(* CoDeSys 2.3.9.55 project: tmeiccoolingskidv2.pro *)
(* Libraries: Standard.lib 20.5.14 01:13:26, Iecsfc.lib 30.1.13 06:05:12, SYSLIBCALLBACK.LIB 30.1.13 06:05:12 *)

(* PLC configuration (modules and I/O channels)
xWaterLow AT %IX10.0 [BOOLOnX_I] Ch_1 Digital input
xWaterLowLow AT %IX10.1 [BOOLOnX_I] Ch_2 Digital input
AT %IX10.2 [BOOLOnX_I] Ch_1 Digital input
AT %IX10.3 [BOOLOnX_I] Ch_2 Digital input
AT %IX10.4 [BOOLOnX_I] Ch_3 Digital input
AT %IX10.5 [BOOLOnX_I] Ch_4 Digital input
0750-0402 4 DI 24 V DC 3.0ms [Type_1_4_Channels] node 2, in %IX10.2 out %QB4
  AT %IX10.6 [BOOLOnX_I] Ch_1 Digital input
  AT %IX10.7 [BOOLOnX_I] Ch_2 Digital input
  AT %IX10.8 [BOOLOnX_I] Ch_3 Digital input
  AT %IX10.9 [BOOLOnX_I] Ch_4 Digital input
xOutput8DO1 AT %QX2.0 [BOOLOnX_Q] Ch_1 Digital output
AT %QX2.1 [BOOLOnX_Q] Ch_2 Digital output
AT %QX2.2 [BOOLOnX_Q] Ch_3 Digital output
AT %QX2.3 [BOOLOnX_Q] Ch_4 Digital output
AT %QX2.4 [BOOLOnX_Q] Ch_5 Digital output
AT %QX2.5 [BOOLOnX_Q] Ch_6 Digital output
AT %QX2.6 [BOOLOnX_Q] Ch_7 Digital output
AT %QX2.7 [BOOLOnX_Q] Ch_8 Digital output
xOutput AT %QX2.8 [BOOLOnX_Q] Ch_1 Digital output
AT %QX2.9 [BOOLOnX_Q] Ch_2 Digital output
AT %QX2.10 [BOOLOnX_Q] Ch_1 Digital output
AT %QX2.11 [BOOLOnX_Q] Ch_2 Digital output
0750-0492 2 AI 4-20mA Diff Measurement Input [Type_8_2_Channels] node 6, in %IB20 out %QB0
  AT %IW0 [WORDOnW_I] Ch_1 Input word
  AT %IW1 [WORDOnW_I] Ch_2 Input word
0750-0461 2 AI PT100 (RTD) [Type_44_2_Channels] node 7, in %IB20 out %QB0
  AT %IW2 [INTOnW_I] Ch_1 signed Input value
  AT %IW3 [INTOnW_I] Ch_2 signed Input value
0750-0461 2 AI PT100 (RTD) [Type_44_2_Channels] node 8, in %IB24 out %QB0
  AT %IW4 [INTOnW_I] Ch_1 signed Input value
  AT %IW5 [INTOnW_I] Ch_2 signed Input value
0750-0455 4 AI 4-20mA s.e. [Type_8_4_Channels] node 9, in %IB28 out %QB0
  AT %IW6 [WORDOnW_I] Ch_1 Input word
  AT %IW7 [WORDOnW_I] Ch_2 Input word
  AT %IW8 [WORDOnW_I] Ch_3 Input word
  AT %IW9 [WORDOnW_I] Ch_4 Input word
0750-0554 2 AO 4-20mA [Type_14_2_Channels] node 10, in %IB32 out %QB0
  AT %QW0 [WORDOnW_Q] Ch_1 Analog output
  AT %QW1 [WORDOnW_Q] Ch_2 Analog output
AT %IX10.10 [BOOLOnX_I] Ch_1 Digital input
AT %IX10.11 [BOOLOnX_I] Ch_2 Digital input
AT %IX10.12 [BOOLOnX_I] Ch_3 Digital input
AT %IX10.13 [BOOLOnX_I] Ch_4 Digital input
Modbus variables [PFC200MODBUS] node 1, in %IB0 out %QB0 {PlcStopBehaviour = 1; FiledbusErrorBehaviour = 1; TcpOperation = 1; TcpPort = 502; TcpTimeout = 600; UdpOperation = 1; UdpPort = 502; RtuOperation = 0; NodeId = 1; ResponseTimeout = 100; Interface = 0; Baud = 115200; StopBits = 1; Parity = 1; FlowCtrl = 0; PhysInterface = 0}
Modbus-Master [MB_MASTER] node 2, in %IB0 out %QB0
*)

(* Global variable list: Global_Variables *)
VAR_GLOBAL
	gaPumps: ARRAY [1..2] OF  ST_PUMP;
	gaTemps: ARRAY [1..3] OF ST_RTD;
	gaSwitches: ARRAY [1..3] OF ST_SWITCH;
	gaFans: ARRAY [1..4] OF ST_FAN;
	gConductivity: ST_COND;
	gFlow: ST_FLOW;
	gAct: ST_ACT;
	gSystem: ST_SYSTEM;
	gcAlarm: INT :=  1;
	gcFault:  INT := 0;
	gTempValCtrlSys: ST_TempValCtrlSys;
	gProgramErrors: ST_ProgramErrors;
	tbFailure: BOOL;
	tbSuccess: BOOL;
	tbTBLog: STRING(256);

	activePump: ST_PUMP;
	standbyPump: ST_PUMP;


END_VAR

(* Data type *)
TYPE HERE :
STRUCT
	On: BOOL;
	Off: BOOL;
	Fault: BOOL;
	Shutting_Down: BOOL;
	Initializing: BOOL;
	Calibrating: BOOL;
	Acknowledge_Fault: BOOL;
	LIST_FLAGS: ARRAY [1..25] OF BOOL;
	System_Active: BOOL;
	PA: BOOL;
	SA: BOOL;

END_STRUCT
END_TYPE

(* Data type in Instrument Data Types *)
TYPE RAWINPUT :
STRUCT
	wRawAnalogWord: WORD;
	iRawAnalogInt: INT;
	xRawDigital: BOOL;
END_STRUCT
END_TYPE

(* Data type *)
TYPE SignalIO :
STRUCT
END_STRUCT
END_TYPE

(* Data type *)
TYPE ST_ACT :
STRUCT
	stDescription: ST_Description;
	stActualization: ST_Analog;
	stCounters: ST_LGCount;
	stCalibrationStatus: ST_CalTest;
	rOpenPerc: REAL; (*Percentage of it being Open*)
END_STRUCT
END_TYPE

(* Data type *)
TYPE ST_ActivePumpStandbyPump :
STRUCT
END_STRUCT
END_TYPE

(* Data type *)
TYPE ST_Analog :
STRUCT
	rGain: REAL;
	rOffset: REAL;
	iRaw: REAL;
	rProcessed: REAL;
END_STRUCT
END_TYPE

(* Data type *)
TYPE ST_Backup :
STRUCT
	xActive: BOOL;
	xRedundant: BOOL;
END_STRUCT
END_TYPE

(* Data type *)
TYPE ST_CalTest :
STRUCT
	xCalibrated: BOOL;
	xTested: BOOL;
END_STRUCT
END_TYPE

(* Data type *)
TYPE ST_COND :
STRUCT
	stDescription: ST_Description;
	stConductivity: ST_Analog; (*Cond Reading Power*)
	stFault: ST_Digital; (*Fault Y/N*)
	stAlarm: ST_DIgital; (*Alarm Y/N*)
	stCounters: ST_LGCount;
	stCalibrationStatus: ST_CalTest;
END_STRUCT
END_TYPE

(* Data type *)
TYPE ST_Count :
STRUCT
	iAlarm: INT;
	iFault: INT;
	iForce: INT;
	iCalibrate: INT;
	iTest: INT;
END_STRUCT
END_TYPE

(* Data type *)
TYPE ST_Description :
STRUCT
	iID : INT;
	iState: INT; (*Offline, Standby,  Active, Calibration, Testing *)
	xFault: BOOL;
	xAlarm: BOOL;
	sDetail:  STRING;
END_STRUCT
END_TYPE

(* Data type *)
TYPE ST_Digital :
STRUCT
	iValue: INT;
END_STRUCT
END_TYPE

(* Data type *)
TYPE ST_FA :
STRUCT
	xFault: BOOL;
	xAlarm: BOOL;
END_STRUCT
END_TYPE

(* Data type *)
TYPE ST_FAN :
STRUCT
	stDescription: ST_Description;
	stActivate: ST_Digital; (*Pump On/Off*)
	stCounters: ST_LGCount;
	stCalibrationStatus: ST_CalTest;
	stBackup: ST_Backup;
END_STRUCT
END_TYPE

(* Data type *)
TYPE ST_FLOW :
STRUCT
	stDescription: ST_Description;
	stFlowRate: ST_Analog; (*Switch Trip*)
	stCounters: ST_LGCount;
	stCalibrationStatus: ST_CalTest;
END_STRUCT
END_TYPE

(* Data type *)
TYPE ST_HeartBeat :
STRUCT
	stDescription: ST_Description;
END_STRUCT
END_TYPE

(* Data type in Instrument Data Types *)
TYPE ST_INST :
STRUCT
	axBoolValues: ARRAY [1..10] OF BOOL;
	aiIntValues: ARRAY [1..10] OF REAL;

END_STRUCT
END_TYPE

(* Data type in Instrument Data Types *)
TYPE ST_INSTRUMENT :
STRUCT
	iState: INT; (*0 = Standby; 1 = Data Loading;*)
	stInput: ST_IO;
	stOutput: ST_IO;
	stMeasurement: ST_MEASUREMENTS;
	stActuateValues: ST_MEASUREMENTS;
END_STRUCT
END_TYPE

(* Data type in Flags *)
TYPE ST_InstrumentFlags :
STRUCT
	xConductivitySensorAlarmTrip: BOOL := FALSE;
	xConductivitySensorFaultTrip: BOOL := FALSE;
	xPump1BadRead: BOOL := FALSE;
	xPump2BadRead: BOOL := FALSE;
	xPump1LPError: BOOL := FALSE;
	xPump2LPError: BOOL := FALSE;
	xConductivitySensorBadRead: BOOL := FALSE;
	xConductivitySensorMisalignment: BOOL := FALSE;
	xConductivitySensorError: BOOL := FALSE;
	xFlowSensorBadRead: BOOL := FALSE;
	xRTD1BadRead: BOOL := FALSE;
	xRTD2BadRead: BOOL := FALSE;
	xRTD3BadRead: BOOL := FALSE;
	xNoPumpBackup: BOOL := FALSE;
	xPump1Failure: BOOL := FALSE;
	xPump2Failure: BOOL := FALSE;
	xRTD1Failure: BOOL := FALSE;
	xRTD2Failure: BOOL := FALSE;
	xRTD3Failure: BOOL := FALSE;
	xConductivitySensorFailure: BOOL := FALSE;
	xFlowSensorFailure: BOOL := FALSE;
	xPressureLow: BOOL := FALSE;
	xPumpPowerLow: BOOL := FALSE;
	xFlowLow: BOOL := FALSE;
	xWaterLevelSensorError: BOOL := FALSE;
END_STRUCT
END_TYPE

(* Data type *)
TYPE ST_IO :
STRUCT
	axDigital: ARRAY [1..100] OF BOOL;
	awAnalog: ARRAY[1..100] OF WORD;
	aiAnalog: ARRAY[1..100] OF INT;
END_STRUCT
END_TYPE

(* Data type *)
TYPE ST_LGCount :
STRUCT
	stLocal : ST_Count;
	stGlobal: ST_Count;
END_STRUCT
END_TYPE

(* Data type in Instrument Data Types *)
TYPE ST_MEASUREMENTS :
STRUCT
	axDigital: ARRAY [1..100] OF BOOL;
	arAnalog: ARRAY[1..100] OF REAL;
END_STRUCT
END_TYPE

(* Data type *)
TYPE ST_PRES :
STRUCT
	stDescription: ST_Description;
	stSwitchTrip: ST_Digital; (*Switch Trip*)
	stCounters: ST_LGCount;
	stCalibrationStatus: ST_CalTest;
END_STRUCT
END_TYPE

(* Data type *)
TYPE ST_ProgramErrors :
STRUCT
	xTempValCtrlSys: BOOL;
	xDataConversion: BOOL;
END_STRUCT
END_TYPE

(* Data type *)
TYPE ST_PUMP :
STRUCT
	stDescription: ST_Description;
	stPumpPower: ST_Analog; (*Pump Power*)
	stActivate: ST_Digital; (*Pump On/Off*)
	stCounters: ST_LGCount;
	stCalibrationStatus: ST_CalTest;
	stBackup: ST_Backup;
END_STRUCT
END_TYPE

(* Data type *)
TYPE ST_RTD :
STRUCT
	stDescription: ST_Description;
	stTempRead: ST_Analog;
	stCounters: ST_LGCount;
	stCalibrationStatus: ST_CalTest;
END_STRUCT
END_TYPE

(* Data type *)
TYPE ST_SPT :
STRUCT
	rSetpoint: REAL;
	rThreshold: REAL;
END_STRUCT
END_TYPE

(* Data type *)
TYPE ST_SWITCH :
STRUCT
	stDescription: ST_Description;
	stSwitchTrip: ST_Digital; (*Switch Trip*)
	stCounters: ST_LGCount;
	stCalibrationStatus: ST_CalTest;
END_STRUCT
END_TYPE

(* Data type *)
TYPE ST_SYSTEM :
STRUCT
	stSystemCounters: ST_SystemCounters;
	stSystemFlags: ST_SystemFlags;
	stInstrumentFlags: ST_instrumentFlags;
	stInputs: ST_SystemInputs;
	stOutputs: ST_SystemOutputs;
END_STRUCT
END_TYPE

(* Data type *)
TYPE ST_SystemCounters :
STRUCT
	iRTDFailures: INT;
	iPumpFailures: INT;
	iActivePump: INT;
	iActiveFanGroup: INT;
END_STRUCT
END_TYPE

(* Data type *)
TYPE ST_SystemFlags :
STRUCT
	xSwitchPumpRequest: BOOL;
	xAwaitInitialization: BOOL;
	xAwaitCalibration: BOOL;
	xFault: BOOL;
	xAlarm: BOOL;
	xPPFError: BOOL;
	xWaterLow: BOOL;
	xWaterVeryLow: BOOL;
END_STRUCT
END_TYPE

(* Data type *)
TYPE ST_SystemInputs :
STRUCT
	rPumpPower: REAL;
	rFlowRate: REAL;
	rConductivity: REAL;
	rTemperature: REAL;
	xPressureLow: BOOL;
	xWaterLow: BOOL;
	xWaterLowLow: BOOL;
	xSystemON: BOOL;
	xConductivityAlarm: BOOL;
	xConductivityFault: BOOL;
END_STRUCT
END_TYPE

(* Data type *)
TYPE ST_SystemMeasurement :
STRUCT

END_STRUCT
END_TYPE

(* Data type *)
TYPE ST_SystemOutputs :
STRUCT
	rValveActuate: REAL;
	xPump1Activate: BOOL;
	xPump2Activate: BOOL;
	xFan12Activate: BOOL;
	xFan34Activate: BOOL;
END_STRUCT
END_TYPE

(* Data type *)
TYPE ST_TempValCtrlSys :
STRUCT
	rDiffThresh: REAL;
	rDiffTol: REAL;
	iSysMeasState: INT;
	xFault: BOOL; (*Fault when all controlers are bad, or program error*)
	xAlarm: BOOL; (*Alarm for fault, when controller is bad, or program error*)
END_STRUCT
END_TYPE

(* POU PLC_PRG, LD *)
PROGRAM PLC_PRG
VAR PERSISTENT
	stPump1: ST_INSTRUMENT;
	stPump2: ST_INSTRUMENT;
	stPump3: ST_INSTRUMENT;
	stRTD1: ST_INSTRUMENT;
	stRTD2: ST_INSTRUMENT;
	stRTD3: ST_INSTRUMENT;
	stFan1: ST_INSTRUMENT;
	stFan2: ST_INSTRUMENT;
	stFan3: ST_INSTRUMENT;
	stFan4: ST_INSTRUMENT;
	stConductivitySensor: ST_INSTRUMENT;
	stFlowSensor: ST_INSTRUMENT;
	stWaterLevelLow: ST_INSTRUMENT;
	stWaterLevelLowLow: ST_INSTRUMENT;
	stPressureLowSensor: ST_INSTRUMENT;
	stSystemRunSwitch: ST_INSTRUMENT;

	stInstrumentFlags: ST_InstrumentFlags;

	stSystem: ST_SYSTEM;
END_VAR
VAR
		xReadAnalog: BOOL;
	xReadTemperature: BOOL;
	fbRunTestBench: RunTestBench;
	xTesting: BOOL;
	xReadDigital: BOOL;
	fbWaterLevelLowCaputer: FB_DigitalCapture;
	fbWaterLevelLowLowCapture: FB_DigitalCapture;
	fbConductivityAlarmCapture: FB_DigitalCapture;
	fbAssignAnalogValues: FB_AssignAnalog;
	fbAAP1: FB_AssignAnalog;
	fbAAP2: FB_AssignAnalog;
	fbAARTD1: FB_AssignAnalog;
	fbAARTD2: FB_AssignAnalog;
	fbAARTD3: FB_AssignAnalog;
	fbAAF3: FB_AssignAnalog;
	fbAAF: FB_AssignAnalog;
	fbAAC: FB_AssignAnalog;
END_VAR
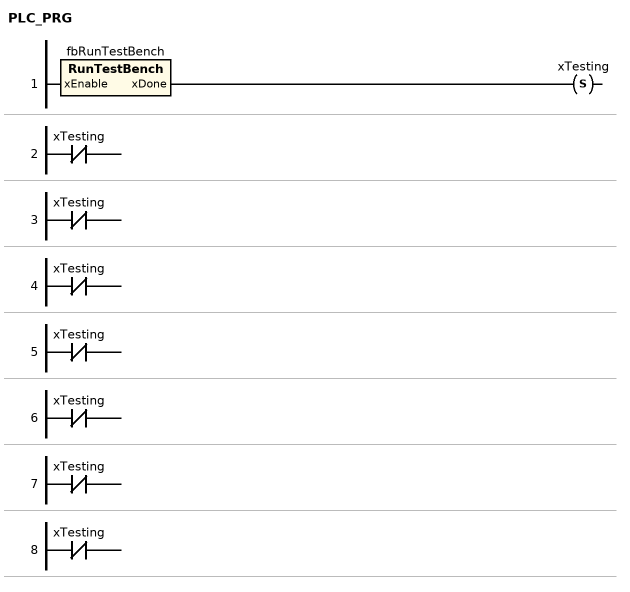
_LD_ (* Ladder Diagram *)
NETWORK 1
	fbRunTestBench:RunTestBench(xEnable: *) --- (S xTesting)
NETWORK 2
	[/xTesting]
NETWORK 3
	[/xTesting]
NETWORK 4
	[/xTesting]
NETWORK 5
	[/xTesting]
NETWORK 6
	[/xTesting]
NETWORK 7
	[/xTesting]
NETWORK 8
	[/xTesting]
_END_LD_
(* the same logic as Structured Text *)
(* Network 1 *)
fbRunTestBench(xEnable := TRUE);
IF fbRunTestBench.xDone THEN xTesting := TRUE; END_IF;
(* Network 2 *)
(* Network 3 *)
(* Network 4 *)
(* Network 5 *)
(* Network 6 *)
(* Network 7 *)
(* Network 8 *)
END_PROGRAM

(* POU RunTestBench, ST *)
FUNCTION_BLOCK RunTestBench
VAR_INPUT
	xEnable: BOOL;
END_VAR
VAR_OUTPUT
	xDone: BOOL := TRUE;
END_VAR
VAR
	istopCase: INT;
	iWait: INT := 0;
END_VAR
IF xEnable = FALSE THEN
	RETURN;
END_IF
TB_MainProgram2();
END_FUNCTION_BLOCK

(* POU TB_MainProgram2, LD *)
PROGRAM TB_MainProgram2
VAR
	PUMP1: ST_INSTRUMENT;
	PUMP2: ST_INSTRUMENT;
	RTD1: ST_INSTRUMENT;
	RTD2: ST_INSTRUMENT;
	RTD3: ST_INSTRUMENT;
	CONDUCTIVITY: ST_INSTRUMENT;
	FLOW: ST_INSTRUMENT;
	WATERLOW: ST_INSTRUMENT;
	WATERLOWLOW: ST_INSTRUMENT;
	PRESSURELOW: ST_INSTRUMENT;
	SYSTEM: ST_SYSTEM;
	main: HERE;
	p1i: WORD := 32768;
	p2i: WORD := 50;
	t1i: INT := 100;
	t2i: INT:= 100;
	t3i: INT:= 100;
	fi: WORD:= 50;
	ci: WORD:= 40;
	wli: BOOL:= FALSE;
	wlli: BOOL:= FALSE;
	cai: BOOL:= FALSE;
	cfi: BOOL:= FALSE;
	pli: BOOL:= FALSE;
	p1mas: REAL:= 32767;
	p2mas: REAL:= 32767;
	t1mas: REAL:= 32767;
	t2mas: REAL:= 32767;
	t3mas: REAL:= 32767;
	fmas: REAL:= 32767;
	cmas: REAL:= 32767;
	p1mis: REAL:= -32768;
	p2mis: REAL:= -32768;
	t1mis: REAL:= 0;
	t2mis: REAL:= 0;
	t3mis: REAL:= 0;
	fmis: REAL:= -32768;
	cmis: REAL:= -32768;
	p1mav: REAL:= 55;
	p2mav: REAL:= 55;
	t1mav: REAL:= 100;
	t2mav: REAL:= 100;
	t3mav: REAL:= 100;
	fmav: REAL:= 20;
	cmaV: REAL:= 2000;
	p1miv: REAL:= 0;
	p2miv: REAL:= 0;
	t1miv: REAL:= 0;
	t2miv: REAL:= 0;
	t3miv: REAL:= 0;
	fmiv: REAL:= 0;
	cmiv: REAL:= 2;
	p1tol: REAL:= 0;
	p2tol: REAL:= 0;
	t1tol: REAL:= 0;
	t2tol: REAL:= 0;
	t3tol: REAL:= 0;
	ftol: REAL:= 0;
	ctol: REAL:=0;
	p1t: TIME:= T#100MS;
	p2t: TIME:= T#100MS;
	t1t: TIME:= T#100MS;
	t2t: TIME:= T#100MS;
	t3t: TIME:= T#100MS;
	ft: TIME:= T#100MS;
	ct: TIME:= T#100MS;
	wlt: TIME:= T#100MS;
	wllt: TIME:= T#100MS;
	cat: TIME:= T#100MS;
	cft: TIME:= T#100MS;
	plt: TIME:= T#100MS;

	p1o: BOOL;
	p2o: BOOL;
	t1o: BOOL;
	t2o: BOOL;
	t3o: BOOL;
	fo: BOOL;
	co: BOOL;
	wlo: BOOL;
	wllo: BOOL;
	cao: BOOL;
	cfo: BOOL;
	plo: BOOL;
	dummy: BOOL;
	fbinstrumentinputscan: FB_InstrumentInputScan;
	fbsysteminstrumentalignment: FB_SystemInstrumentAlignment;
	fbcheckwaterlevel: FB_CheckWaterLevel;
	fbcheckconductivity: FB_CheckConductivity;
	fbpowerpressureflowthreshold: FB_PowerPressureFlowThreshold;
	fbpowerpressureflowvote: FB_PowerPressureFlowVote;
	fbpumpstartswitchroutine: FB_PumpStartSwitchRoutine;
	xsysalrm1: BOOL;
	xsysfault1: BOOL;
	xsysalarm2: BOOL;
	xsysfault3: BOOL;
	xsysfault2: BOOL;
		xsysalarm3: BOOL;
		xsysalarm4: BOOL;
		xsysfault4: BOOL;
		xpumpswitchrequest2: BOOL;
		xpumpswitchrequest1: BOOL;
		xSystemRun: BOOL;
		xStartDelay: BOOL;
		startdelaytimer: TON;
		fbtempboundcheck: FB_TemperatureBoundCheck;
		xsysalarm5: BOOL;
	xsysfault5: BOOL;
	fbsysstart: FB_SystemStart;
	fbfaultcheck: FB_FaultCheck;
	fbstop: FB_SystemStop;
	fbpumpcontrol: FB_PumpControl;
END_VAR
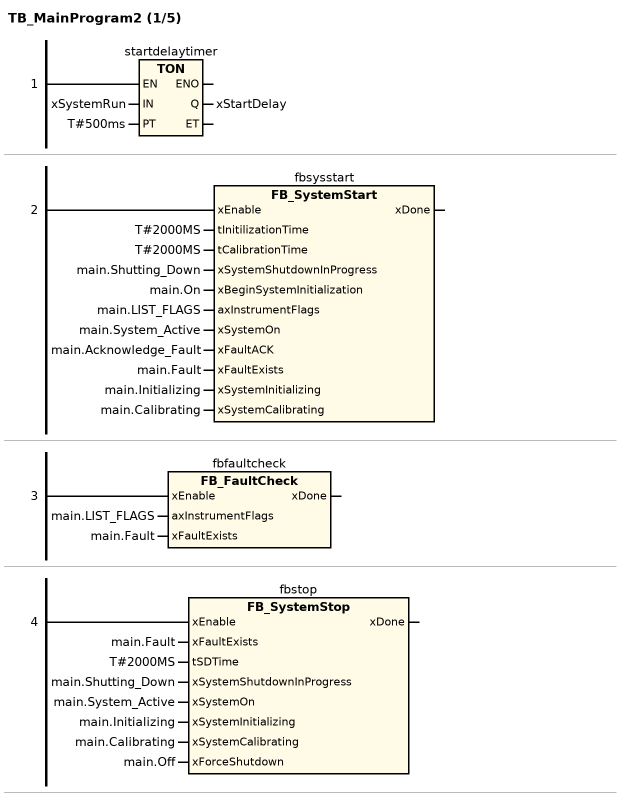
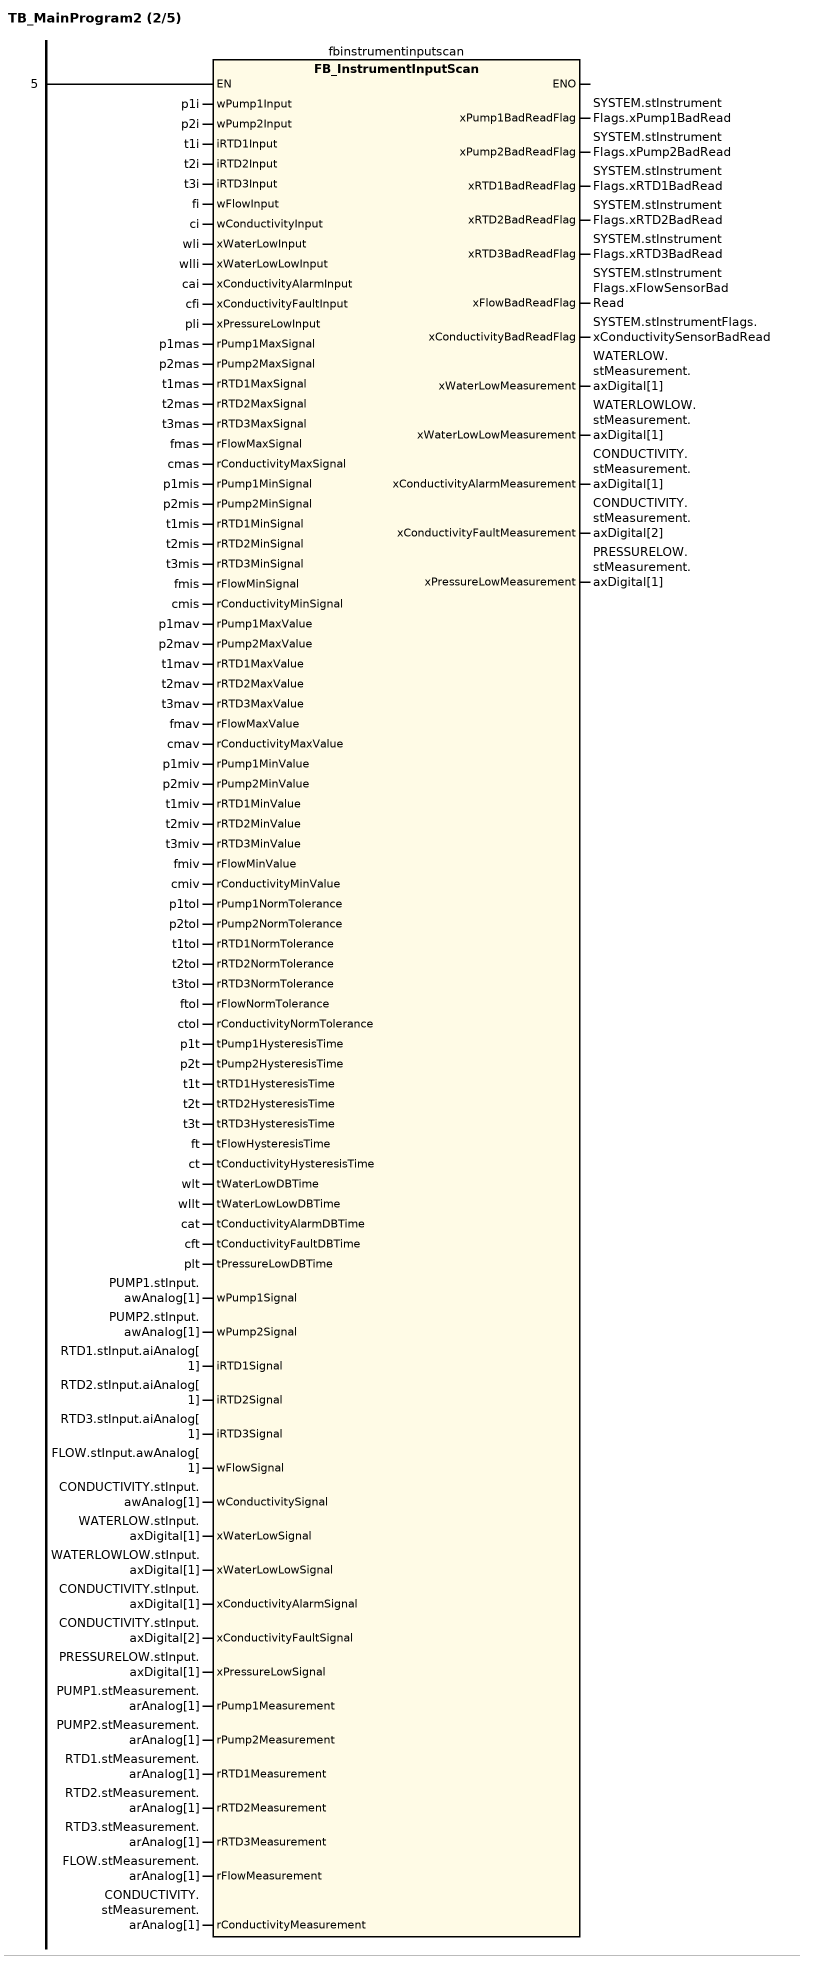
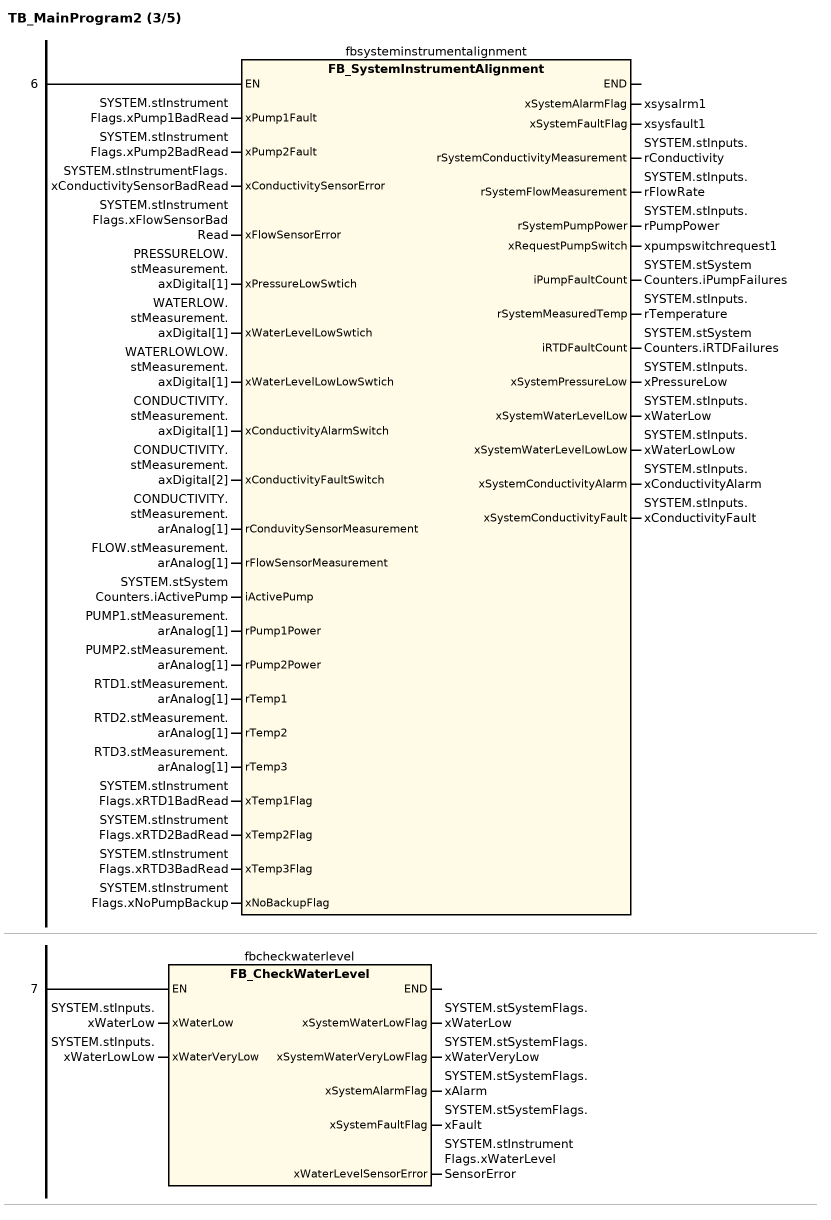
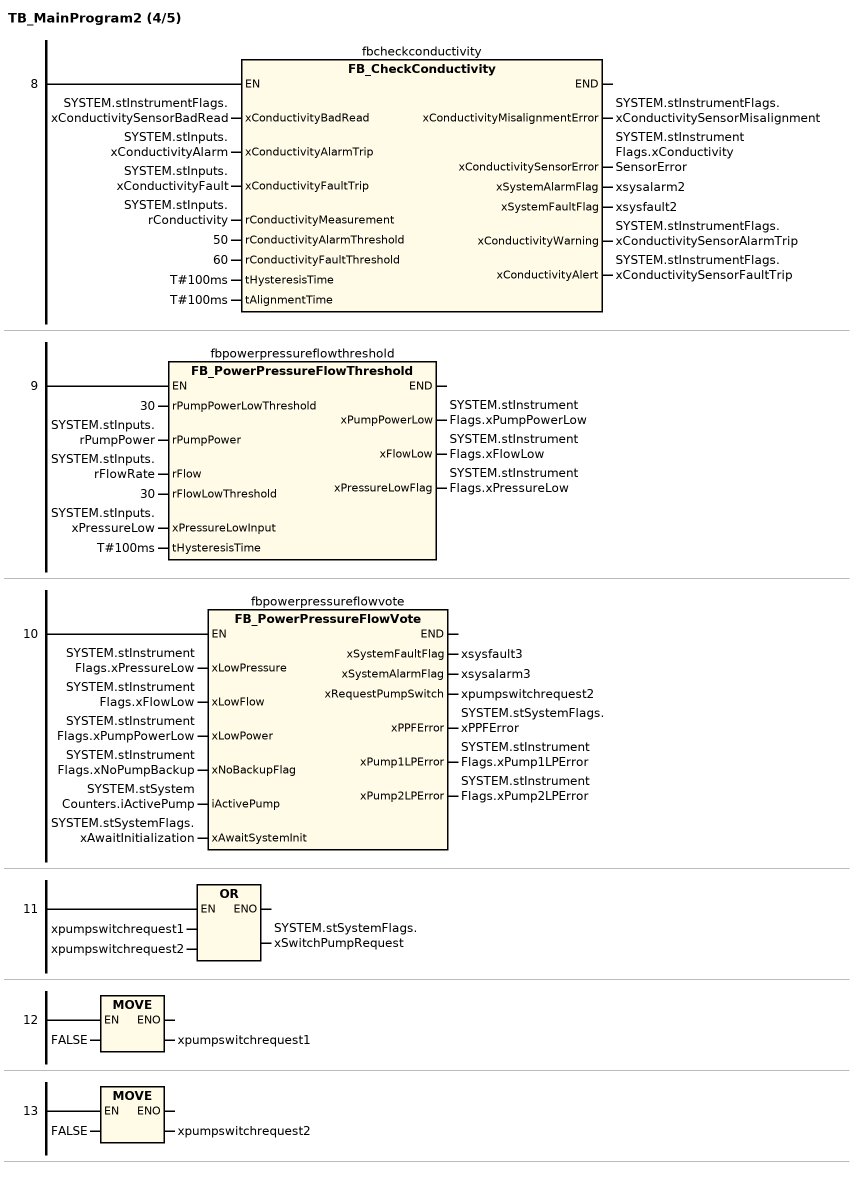
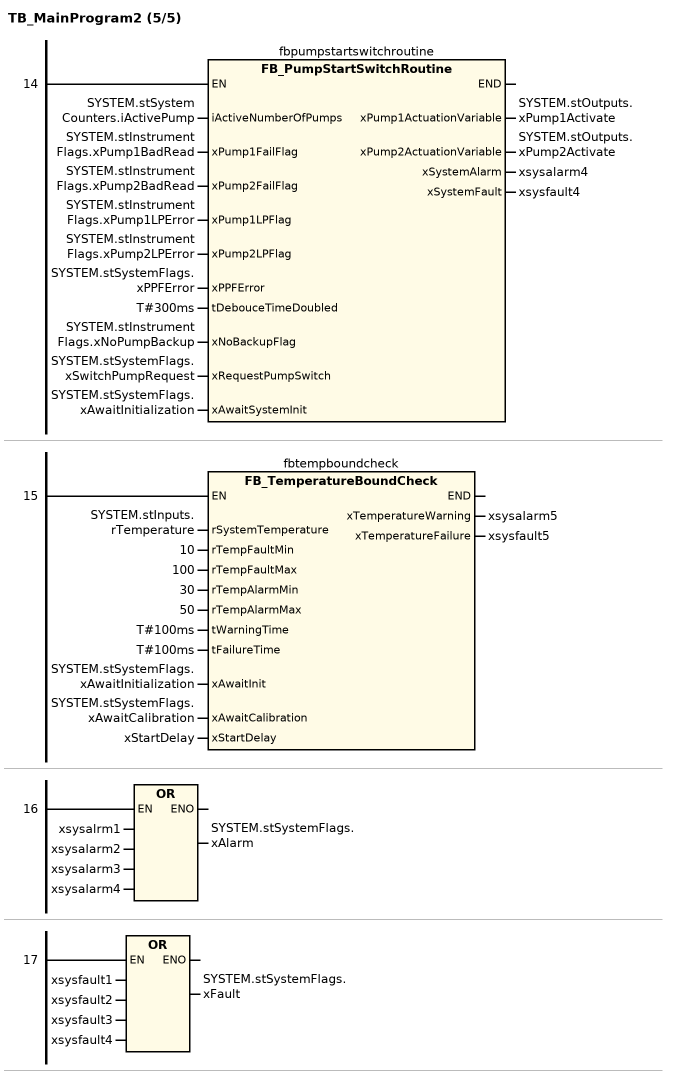
_LD_ (* Ladder Diagram *)
NETWORK 1
	*
		EN --- startdelaytimer:TON(IN: xSystemRun, PT: T#500ms) => xStartDelay
NETWORK 2
	fbsysstart:FB_SystemStart(xEnable: *, tInitilizationTime: T#2000MS, tCalibrationTime: T#2000MS, xSystemShutdownInProgress: main.Shutting_Down, xBeginSystemInitialization: main.On, axInstrumentFlags: main.LIST_FLAGS, xSystemOn: main.System_Active, xFaultACK: main.Acknowledge_Fault, xFaultExists: main.Fault, xSystemInitializing: main.Initializing, xSystemCalibrating: main.Calibrating)
NETWORK 3
	fbfaultcheck:FB_FaultCheck(xEnable: *, axInstrumentFlags: main.LIST_FLAGS, xFaultExists: main.Fault)
NETWORK 4
	fbstop:FB_SystemStop(xEnable: *, xFaultExists: main.Fault, tSDTime: T#2000MS, xSystemShutdownInProgress: main.Shutting_Down, xSystemOn: main.System_Active, xSystemInitializing: main.Initializing, xSystemCalibrating: main.Calibrating, xForceShutdown: main.Off)
NETWORK 5
	*
		EN --- fbinstrumentinputscan:FB_InstrumentInputScan(wPump1Input: p1i, wPump2Input: p2i, iRTD1Input: t1i, iRTD2Input: t2i, iRTD3Input: t3i, wFlowInput: fi, wConductivityInput: ci, xWaterLowInput: wli, xWaterLowLowInput: wlli, xConductivityAlarmInput: cai, xConductivityFaultInput: cfi, xPressureLowInput: pli, rPump1MaxSignal: p1mas, rPump2MaxSignal: p2mas, rRTD1MaxSignal: t1mas, rRTD2MaxSignal: t2mas, rRTD3MaxSignal: t3mas, rFlowMaxSignal: fmas, rConductivityMaxSignal: cmas, rPump1MinSignal: p1mis, rPump2MinSignal: p2mis, rRTD1MinSignal: t1mis, rRTD2MinSignal: t2mis, rRTD3MinSignal: t3mis, rFlowMinSignal: fmis, rConductivityMinSignal: cmis, rPump1MaxValue: p1mav, rPump2MaxValue: p2mav, rRTD1MaxValue: t1mav, rRTD2MaxValue: t2mav, rRTD3MaxValue: t3mav, rFlowMaxValue: fmav, rConductivityMaxValue: cmav, rPump1MinValue: p1miv, rPump2MinValue: p2miv, rRTD1MinValue: t1miv, rRTD2MinValue: t2miv, rRTD3MinValue: t3miv, rFlowMinValue: fmiv, rConductivityMinValue: cmiv, rPump1NormTolerance: p1tol, rPump2NormTolerance: p2tol, rRTD1NormTolerance: t1tol, rRTD2NormTolerance: t2tol, rRTD3NormTolerance: t3tol, rFlowNormTolerance: ftol, rConductivityNormTolerance: ctol, tPump1HysteresisTime: p1t, tPump2HysteresisTime: p2t, tRTD1HysteresisTime: t1t, tRTD2HysteresisTime: t2t, tRTD3HysteresisTime: t3t, tFlowHysteresisTime: ft, tConductivityHysteresisTime: ct, tWaterLowDBTime: wlt, tWaterLowLowDBTime: wllt, tConductivityAlarmDBTime: cat, tConductivityFaultDBTime: cft, tPressureLowDBTime: plt, wPump1Signal: PUMP1.stInput.awAnalog[1], wPump2Signal: PUMP2.stInput.awAnalog[1], iRTD1Signal: RTD1.stInput.aiAnalog[1], iRTD2Signal: RTD2.stInput.aiAnalog[1], iRTD3Signal: RTD3.stInput.aiAnalog[1], wFlowSignal: FLOW.stInput.awAnalog[1], wConductivitySignal: CONDUCTIVITY.stInput.awAnalog[1], xWaterLowSignal: WATERLOW.stInput.axDigital[1], xWaterLowLowSignal: WATERLOWLOW.stInput.axDigital[1], xConductivityAlarmSignal: CONDUCTIVITY.stInput.axDigital[1], xConductivityFaultSignal: CONDUCTIVITY.stInput.axDigital[2], xPressureLowSignal: PRESSURELOW.stInput.axDigital[1], rPump1Measurement: PUMP1.stMeasurement.arAnalog[1], rPump2Measurement: PUMP2.stMeasurement.arAnalog[1], rRTD1Measurement: RTD1.stMeasurement.arAnalog[1], rRTD2Measurement: RTD2.stMeasurement.arAnalog[1], rRTD3Measurement: RTD3.stMeasurement.arAnalog[1], rFlowMeasurement: FLOW.stMeasurement.arAnalog[1], rConductivityMeasurement: CONDUCTIVITY.stMeasurement.arAnalog[1], xPump2BadReadFlag => SYSTEM.stInstrumentFlags.xPump2BadRead, xRTD1BadReadFlag => SYSTEM.stInstrumentFlags.xRTD1BadRead, xRTD2BadReadFlag => SYSTEM.stInstrumentFlags.xRTD2BadRead, xRTD3BadReadFlag => SYSTEM.stInstrumentFlags.xRTD3BadRead, xFlowBadReadFlag => SYSTEM.stInstrumentFlags.xFlowSensorBadRead, xConductivityBadReadFlag => SYSTEM.stInstrumentFlags.xConductivitySensorBadRead, xWaterLowMeasurement => WATERLOW.stMeasurement.axDigital[1], xWaterLowLowMeasurement => WATERLOWLOW.stMeasurement.axDigital[1], xConductivityAlarmMeasurement => CONDUCTIVITY.stMeasurement.axDigital[1], xConductivityFaultMeasurement => CONDUCTIVITY.stMeasurement.axDigital[2], xPressureLowMeasurement => PRESSURELOW.stMeasurement.axDigital[1]) => SYSTEM.stInstrumentFlags.xPump1BadRead
NETWORK 6
	fbsysteminstrumentalignment:FB_SystemInstrumentAlignment(EN: *, xPump1Fault: SYSTEM.stInstrumentFlags.xPump1BadRead, xPump2Fault: SYSTEM.stInstrumentFlags.xPump2BadRead, xConductivitySensorError: SYSTEM.stInstrumentFlags.xConductivitySensorBadRead, xFlowSensorError: SYSTEM.stInstrumentFlags.xFlowSensorBadRead, xPressureLowSwtich: PRESSURELOW.stMeasurement.axDigital[1], xWaterLevelLowSwtich: WATERLOW.stMeasurement.axDigital[1], xWaterLevelLowLowSwtich: WATERLOWLOW.stMeasurement.axDigital[1], xConductivityAlarmSwitch: CONDUCTIVITY.stMeasurement.axDigital[1], xConductivityFaultSwitch: CONDUCTIVITY.stMeasurement.axDigital[2], rConduvitySensorMeasurement: CONDUCTIVITY.stMeasurement.arAnalog[1], rFlowSensorMeasurement: FLOW.stMeasurement.arAnalog[1], iActivePump: SYSTEM.stSystemCounters.iActivePump, rPump1Power: PUMP1.stMeasurement.arAnalog[1], rPump2Power: PUMP2.stMeasurement.arAnalog[1], rTemp1: RTD1.stMeasurement.arAnalog[1], rTemp2: RTD2.stMeasurement.arAnalog[1], rTemp3: RTD3.stMeasurement.arAnalog[1], xTemp1Flag: SYSTEM.stInstrumentFlags.xRTD1BadRead, xTemp2Flag: SYSTEM.stInstrumentFlags.xRTD2BadRead, xTemp3Flag: SYSTEM.stInstrumentFlags.xRTD3BadRead, xNoBackupFlag: SYSTEM.stInstrumentFlags.xNoPumpBackup, xSystemAlarmFlag => xsysalrm1, xSystemFaultFlag => xsysfault1, rSystemConductivityMeasurement => SYSTEM.stInputs.rConductivity, rSystemFlowMeasurement => SYSTEM.stInputs.rFlowRate, rSystemPumpPower => SYSTEM.stInputs.rPumpPower, xRequestPumpSwitch => xpumpswitchrequest1, iPumpFaultCount => SYSTEM.stSystemCounters.iPumpFailures, rSystemMeasuredTemp => SYSTEM.stInputs.rTemperature, iRTDFaultCount => SYSTEM.stSystemCounters.iRTDFailures, xSystemPressureLow => SYSTEM.stInputs.xPressureLow, xSystemWaterLevelLow => SYSTEM.stInputs.xWaterLow, xSystemWaterLevelLowLow => SYSTEM.stInputs.xWaterLowLow, xSystemConductivityAlarm => SYSTEM.stInputs.xConductivityAlarm, xSystemConductivityFault => SYSTEM.stInputs.xConductivityFault)
NETWORK 7
	fbcheckwaterlevel:FB_CheckWaterLevel(EN: *, xWaterLow: SYSTEM.stInputs.xWaterLow, xWaterVeryLow: SYSTEM.stInputs.xWaterLowLow, xSystemWaterLowFlag => SYSTEM.stSystemFlags.xWaterLow, xSystemWaterVeryLowFlag => SYSTEM.stSystemFlags.xWaterVeryLow, xSystemAlarmFlag => SYSTEM.stSystemFlags.xAlarm, xSystemFaultFlag => SYSTEM.stSystemFlags.xFault, xWaterLevelSensorError => SYSTEM.stInstrumentFlags.xWaterLevelSensorError)
NETWORK 8
	fbcheckconductivity:FB_CheckConductivity(EN: *, xConductivityBadRead: SYSTEM.stInstrumentFlags.xConductivitySensorBadRead, xConductivityAlarmTrip: SYSTEM.stInputs.xConductivityAlarm, xConductivityFaultTrip: SYSTEM.stInputs.xConductivityFault, rConductivityMeasurement: SYSTEM.stInputs.rConductivity, rConductivityAlarmThreshold: 50, rConductivityFaultThreshold: 60, tHysteresisTime: T#100ms, tAlignmentTime: T#100ms, xConductivityMisalignmentError => SYSTEM.stInstrumentFlags.xConductivitySensorMisalignment, xConductivitySensorError => SYSTEM.stInstrumentFlags.xConductivitySensorError, xSystemAlarmFlag => xsysalarm2, xSystemFaultFlag => xsysfault2, xConductivityWarning => SYSTEM.stInstrumentFlags.xConductivitySensorAlarmTrip, xConductivityAlert => SYSTEM.stInstrumentFlags.xConductivitySensorFaultTrip)
NETWORK 9
	fbpowerpressureflowthreshold:FB_PowerPressureFlowThreshold(EN: *, rPumpPowerLowThreshold: 30, rPumpPower: SYSTEM.stInputs.rPumpPower, rFlow: SYSTEM.stInputs.rFlowRate, rFlowLowThreshold: 30, xPressureLowInput: SYSTEM.stInputs.xPressureLow, tHysteresisTime: T#100ms, xPumpPowerLow => SYSTEM.stInstrumentFlags.xPumpPowerLow, xFlowLow => SYSTEM.stInstrumentFlags.xFlowLow, xPressureLowFlag => SYSTEM.stInstrumentFlags.xPressureLow)
NETWORK 10
	fbpowerpressureflowvote:FB_PowerPressureFlowVote(EN: *, xLowPressure: SYSTEM.stInstrumentFlags.xPressureLow, xLowFlow: SYSTEM.stInstrumentFlags.xFlowLow, xLowPower: SYSTEM.stInstrumentFlags.xPumpPowerLow, xNoBackupFlag: SYSTEM.stInstrumentFlags.xNoPumpBackup, iActivePump: SYSTEM.stSystemCounters.iActivePump, xAwaitSystemInit: SYSTEM.stSystemFlags.xAwaitInitialization, xSystemFaultFlag => xsysfault3, xSystemAlarmFlag => xsysalarm3, xRequestPumpSwitch => xpumpswitchrequest2, xPPFError => SYSTEM.stSystemFlags.xPPFError, xPump1LPError => SYSTEM.stInstrumentFlags.xPump1LPError, xPump2LPError => SYSTEM.stInstrumentFlags.xPump2LPError)
NETWORK 11
	*
		EN --- OR(xpumpswitchrequest1, xpumpswitchrequest2) => SYSTEM.stSystemFlags.xSwitchPumpRequest
NETWORK 12
	*
		EN --- MOVE(FALSE) => xpumpswitchrequest1
NETWORK 13
	*
		EN --- MOVE(FALSE) => xpumpswitchrequest2
NETWORK 14
	fbpumpstartswitchroutine:FB_PumpStartSwitchRoutine(EN: *, iActiveNumberOfPumps: SYSTEM.stSystemCounters.iActivePump, xPump1FailFlag: SYSTEM.stInstrumentFlags.xPump1BadRead, xPump2FailFlag: SYSTEM.stInstrumentFlags.xPump2BadRead, xPump1LPFlag: SYSTEM.stInstrumentFlags.xPump1LPError, xPump2LPFlag: SYSTEM.stInstrumentFlags.xPump2LPError, xPPFError: SYSTEM.stSystemFlags.xPPFError, tDebouceTimeDoubled: T#300ms, xNoBackupFlag: SYSTEM.stInstrumentFlags.xNoPumpBackup, xRequestPumpSwitch: SYSTEM.stSystemFlags.xSwitchPumpRequest, xAwaitSystemInit: SYSTEM.stSystemFlags.xAwaitInitialization, xPump1ActuationVariable => SYSTEM.stOutputs.xPump1Activate, xPump2ActuationVariable => SYSTEM.stOutputs.xPump2Activate, xSystemAlarm => xsysalarm4, xSystemFault => xsysfault4)
NETWORK 15
	fbtempboundcheck:FB_TemperatureBoundCheck(EN: *, rSystemTemperature: SYSTEM.stInputs.rTemperature, rTempFaultMin: 10, rTempFaultMax: 100, rTempAlarmMin: 30, rTempAlarmMax: 50, tWarningTime: T#100ms, tFailureTime: T#100ms, xAwaitInit: SYSTEM.stSystemFlags.xAwaitInitialization, xAwaitCalibration: SYSTEM.stSystemFlags.xAwaitCalibration, xStartDelay: xStartDelay, xTemperatureWarning => xsysalarm5, xTemperatureFailure => xsysfault5)
NETWORK 16
	*
		EN --- OR(xsysalrm1, xsysalarm2, xsysalarm3, xsysalarm4) => SYSTEM.stSystemFlags.xAlarm
NETWORK 17
	*
		EN --- OR(xsysfault1, xsysfault2, xsysfault3, xsysfault4) => SYSTEM.stSystemFlags.xFault
_END_LD_
(* the same logic as Structured Text *)
(* Network 1 *)
startdelaytimer(IN := xSystemRun, PT := T#500ms);
xStartDelay := startdelaytimer.Q;
(* Network 2 *)
fbsysstart(xEnable := TRUE, tInitilizationTime := T#2000MS, tCalibrationTime := T#2000MS, xSystemShutdownInProgress := main.Shutting_Down, xBeginSystemInitialization := main.On, axInstrumentFlags := main.LIST_FLAGS, xSystemOn := main.System_Active, xFaultACK := main.Acknowledge_Fault, xFaultExists := main.Fault, xSystemInitializing := main.Initializing, xSystemCalibrating := main.Calibrating);
(* Network 3 *)
fbfaultcheck(xEnable := TRUE, axInstrumentFlags := main.LIST_FLAGS, xFaultExists := main.Fault);
(* Network 4 *)
fbstop(xEnable := TRUE, xFaultExists := main.Fault, tSDTime := T#2000MS, xSystemShutdownInProgress := main.Shutting_Down, xSystemOn := main.System_Active, xSystemInitializing := main.Initializing, xSystemCalibrating := main.Calibrating, xForceShutdown := main.Off);
(* Network 5 *)
fbinstrumentinputscan(wPump1Input := p1i, wPump2Input := p2i, iRTD1Input := t1i, iRTD2Input := t2i, iRTD3Input := t3i, wFlowInput := fi, wConductivityInput := ci, xWaterLowInput := wli, xWaterLowLowInput := wlli, xConductivityAlarmInput := cai, xConductivityFaultInput := cfi, xPressureLowInput := pli, rPump1MaxSignal := p1mas, rPump2MaxSignal := p2mas, rRTD1MaxSignal := t1mas, rRTD2MaxSignal := t2mas, rRTD3MaxSignal := t3mas, rFlowMaxSignal := fmas, rConductivityMaxSignal := cmas, rPump1MinSignal := p1mis, rPump2MinSignal := p2mis, rRTD1MinSignal := t1mis, rRTD2MinSignal := t2mis, rRTD3MinSignal := t3mis, rFlowMinSignal := fmis, rConductivityMinSignal := cmis, rPump1MaxValue := p1mav, rPump2MaxValue := p2mav, rRTD1MaxValue := t1mav, rRTD2MaxValue := t2mav, rRTD3MaxValue := t3mav, rFlowMaxValue := fmav, rConductivityMaxValue := cmav, rPump1MinValue := p1miv, rPump2MinValue := p2miv, rRTD1MinValue := t1miv, rRTD2MinValue := t2miv, rRTD3MinValue := t3miv, rFlowMinValue := fmiv, rConductivityMinValue := cmiv, rPump1NormTolerance := p1tol, rPump2NormTolerance := p2tol, rRTD1NormTolerance := t1tol, rRTD2NormTolerance := t2tol, rRTD3NormTolerance := t3tol, rFlowNormTolerance := ftol, rConductivityNormTolerance := ctol, tPump1HysteresisTime := p1t, tPump2HysteresisTime := p2t, tRTD1HysteresisTime := t1t, tRTD2HysteresisTime := t2t, tRTD3HysteresisTime := t3t, tFlowHysteresisTime := ft, tConductivityHysteresisTime := ct, tWaterLowDBTime := wlt, tWaterLowLowDBTime := wllt, tConductivityAlarmDBTime := cat, tConductivityFaultDBTime := cft, tPressureLowDBTime := plt, wPump1Signal := PUMP1.stInput.awAnalog[1], wPump2Signal := PUMP2.stInput.awAnalog[1], iRTD1Signal := RTD1.stInput.aiAnalog[1], iRTD2Signal := RTD2.stInput.aiAnalog[1], iRTD3Signal := RTD3.stInput.aiAnalog[1], wFlowSignal := FLOW.stInput.awAnalog[1], wConductivitySignal := CONDUCTIVITY.stInput.awAnalog[1], xWaterLowSignal := WATERLOW.stInput.axDigital[1], xWaterLowLowSignal := WATERLOWLOW.stInput.axDigital[1], xConductivityAlarmSignal := CONDUCTIVITY.stInput.axDigital[1], xConductivityFaultSignal := CONDUCTIVITY.stInput.axDigital[2], xPressureLowSignal := PRESSURELOW.stInput.axDigital[1], rPump1Measurement := PUMP1.stMeasurement.arAnalog[1], rPump2Measurement := PUMP2.stMeasurement.arAnalog[1], rRTD1Measurement := RTD1.stMeasurement.arAnalog[1], rRTD2Measurement := RTD2.stMeasurement.arAnalog[1], rRTD3Measurement := RTD3.stMeasurement.arAnalog[1], rFlowMeasurement := FLOW.stMeasurement.arAnalog[1], rConductivityMeasurement := CONDUCTIVITY.stMeasurement.arAnalog[1]);
SYSTEM.stInstrumentFlags.xPump2BadRead := fbinstrumentinputscan.xPump2BadReadFlag;
SYSTEM.stInstrumentFlags.xRTD1BadRead := fbinstrumentinputscan.xRTD1BadReadFlag;
SYSTEM.stInstrumentFlags.xRTD2BadRead := fbinstrumentinputscan.xRTD2BadReadFlag;
SYSTEM.stInstrumentFlags.xRTD3BadRead := fbinstrumentinputscan.xRTD3BadReadFlag;
SYSTEM.stInstrumentFlags.xFlowSensorBadRead := fbinstrumentinputscan.xFlowBadReadFlag;
SYSTEM.stInstrumentFlags.xConductivitySensorBadRead := fbinstrumentinputscan.xConductivityBadReadFlag;
WATERLOW.stMeasurement.axDigital[1] := fbinstrumentinputscan.xWaterLowMeasurement;
WATERLOWLOW.stMeasurement.axDigital[1] := fbinstrumentinputscan.xWaterLowLowMeasurement;
CONDUCTIVITY.stMeasurement.axDigital[1] := fbinstrumentinputscan.xConductivityAlarmMeasurement;
CONDUCTIVITY.stMeasurement.axDigital[2] := fbinstrumentinputscan.xConductivityFaultMeasurement;
PRESSURELOW.stMeasurement.axDigital[1] := fbinstrumentinputscan.xPressureLowMeasurement;
SYSTEM.stInstrumentFlags.xPump1BadRead := fbinstrumentinputscan.xPump1BadReadFlag;
(* Network 6 *)
fbsysteminstrumentalignment(EN := TRUE, xPump1Fault := SYSTEM.stInstrumentFlags.xPump1BadRead, xPump2Fault := SYSTEM.stInstrumentFlags.xPump2BadRead, xConductivitySensorError := SYSTEM.stInstrumentFlags.xConductivitySensorBadRead, xFlowSensorError := SYSTEM.stInstrumentFlags.xFlowSensorBadRead, xPressureLowSwtich := PRESSURELOW.stMeasurement.axDigital[1], xWaterLevelLowSwtich := WATERLOW.stMeasurement.axDigital[1], xWaterLevelLowLowSwtich := WATERLOWLOW.stMeasurement.axDigital[1], xConductivityAlarmSwitch := CONDUCTIVITY.stMeasurement.axDigital[1], xConductivityFaultSwitch := CONDUCTIVITY.stMeasurement.axDigital[2], rConduvitySensorMeasurement := CONDUCTIVITY.stMeasurement.arAnalog[1], rFlowSensorMeasurement := FLOW.stMeasurement.arAnalog[1], iActivePump := SYSTEM.stSystemCounters.iActivePump, rPump1Power := PUMP1.stMeasurement.arAnalog[1], rPump2Power := PUMP2.stMeasurement.arAnalog[1], rTemp1 := RTD1.stMeasurement.arAnalog[1], rTemp2 := RTD2.stMeasurement.arAnalog[1], rTemp3 := RTD3.stMeasurement.arAnalog[1], xTemp1Flag := SYSTEM.stInstrumentFlags.xRTD1BadRead, xTemp2Flag := SYSTEM.stInstrumentFlags.xRTD2BadRead, xTemp3Flag := SYSTEM.stInstrumentFlags.xRTD3BadRead, xNoBackupFlag := SYSTEM.stInstrumentFlags.xNoPumpBackup);
xsysalrm1 := fbsysteminstrumentalignment.xSystemAlarmFlag;
xsysfault1 := fbsysteminstrumentalignment.xSystemFaultFlag;
SYSTEM.stInputs.rConductivity := fbsysteminstrumentalignment.rSystemConductivityMeasurement;
SYSTEM.stInputs.rFlowRate := fbsysteminstrumentalignment.rSystemFlowMeasurement;
SYSTEM.stInputs.rPumpPower := fbsysteminstrumentalignment.rSystemPumpPower;
xpumpswitchrequest1 := fbsysteminstrumentalignment.xRequestPumpSwitch;
SYSTEM.stSystemCounters.iPumpFailures := fbsysteminstrumentalignment.iPumpFaultCount;
SYSTEM.stInputs.rTemperature := fbsysteminstrumentalignment.rSystemMeasuredTemp;
SYSTEM.stSystemCounters.iRTDFailures := fbsysteminstrumentalignment.iRTDFaultCount;
SYSTEM.stInputs.xPressureLow := fbsysteminstrumentalignment.xSystemPressureLow;
SYSTEM.stInputs.xWaterLow := fbsysteminstrumentalignment.xSystemWaterLevelLow;
SYSTEM.stInputs.xWaterLowLow := fbsysteminstrumentalignment.xSystemWaterLevelLowLow;
SYSTEM.stInputs.xConductivityAlarm := fbsysteminstrumentalignment.xSystemConductivityAlarm;
SYSTEM.stInputs.xConductivityFault := fbsysteminstrumentalignment.xSystemConductivityFault;
(* Network 7 *)
fbcheckwaterlevel(EN := TRUE, xWaterLow := SYSTEM.stInputs.xWaterLow, xWaterVeryLow := SYSTEM.stInputs.xWaterLowLow);
SYSTEM.stSystemFlags.xWaterLow := fbcheckwaterlevel.xSystemWaterLowFlag;
SYSTEM.stSystemFlags.xWaterVeryLow := fbcheckwaterlevel.xSystemWaterVeryLowFlag;
SYSTEM.stSystemFlags.xAlarm := fbcheckwaterlevel.xSystemAlarmFlag;
SYSTEM.stSystemFlags.xFault := fbcheckwaterlevel.xSystemFaultFlag;
SYSTEM.stInstrumentFlags.xWaterLevelSensorError := fbcheckwaterlevel.xWaterLevelSensorError;
(* Network 8 *)
fbcheckconductivity(EN := TRUE, xConductivityBadRead := SYSTEM.stInstrumentFlags.xConductivitySensorBadRead, xConductivityAlarmTrip := SYSTEM.stInputs.xConductivityAlarm, xConductivityFaultTrip := SYSTEM.stInputs.xConductivityFault, rConductivityMeasurement := SYSTEM.stInputs.rConductivity, rConductivityAlarmThreshold := 50, rConductivityFaultThreshold := 60, tHysteresisTime := T#100ms, tAlignmentTime := T#100ms);
SYSTEM.stInstrumentFlags.xConductivitySensorMisalignment := fbcheckconductivity.xConductivityMisalignmentError;
SYSTEM.stInstrumentFlags.xConductivitySensorError := fbcheckconductivity.xConductivitySensorError;
xsysalarm2 := fbcheckconductivity.xSystemAlarmFlag;
xsysfault2 := fbcheckconductivity.xSystemFaultFlag;
SYSTEM.stInstrumentFlags.xConductivitySensorAlarmTrip := fbcheckconductivity.xConductivityWarning;
SYSTEM.stInstrumentFlags.xConductivitySensorFaultTrip := fbcheckconductivity.xConductivityAlert;
(* Network 9 *)
fbpowerpressureflowthreshold(EN := TRUE, rPumpPowerLowThreshold := 30, rPumpPower := SYSTEM.stInputs.rPumpPower, rFlow := SYSTEM.stInputs.rFlowRate, rFlowLowThreshold := 30, xPressureLowInput := SYSTEM.stInputs.xPressureLow, tHysteresisTime := T#100ms);
SYSTEM.stInstrumentFlags.xPumpPowerLow := fbpowerpressureflowthreshold.xPumpPowerLow;
SYSTEM.stInstrumentFlags.xFlowLow := fbpowerpressureflowthreshold.xFlowLow;
SYSTEM.stInstrumentFlags.xPressureLow := fbpowerpressureflowthreshold.xPressureLowFlag;
(* Network 10 *)
fbpowerpressureflowvote(EN := TRUE, xLowPressure := SYSTEM.stInstrumentFlags.xPressureLow, xLowFlow := SYSTEM.stInstrumentFlags.xFlowLow, xLowPower := SYSTEM.stInstrumentFlags.xPumpPowerLow, xNoBackupFlag := SYSTEM.stInstrumentFlags.xNoPumpBackup, iActivePump := SYSTEM.stSystemCounters.iActivePump, xAwaitSystemInit := SYSTEM.stSystemFlags.xAwaitInitialization);
xsysfault3 := fbpowerpressureflowvote.xSystemFaultFlag;
xsysalarm3 := fbpowerpressureflowvote.xSystemAlarmFlag;
xpumpswitchrequest2 := fbpowerpressureflowvote.xRequestPumpSwitch;
SYSTEM.stSystemFlags.xPPFError := fbpowerpressureflowvote.xPPFError;
SYSTEM.stInstrumentFlags.xPump1LPError := fbpowerpressureflowvote.xPump1LPError;
SYSTEM.stInstrumentFlags.xPump2LPError := fbpowerpressureflowvote.xPump2LPError;
(* Network 11 *)
SYSTEM.stSystemFlags.xSwitchPumpRequest := xpumpswitchrequest1 OR xpumpswitchrequest2;
(* Network 12 *)
xpumpswitchrequest1 := FALSE;
(* Network 13 *)
xpumpswitchrequest2 := FALSE;
(* Network 14 *)
fbpumpstartswitchroutine(EN := TRUE, iActiveNumberOfPumps := SYSTEM.stSystemCounters.iActivePump, xPump1FailFlag := SYSTEM.stInstrumentFlags.xPump1BadRead, xPump2FailFlag := SYSTEM.stInstrumentFlags.xPump2BadRead, xPump1LPFlag := SYSTEM.stInstrumentFlags.xPump1LPError, xPump2LPFlag := SYSTEM.stInstrumentFlags.xPump2LPError, xPPFError := SYSTEM.stSystemFlags.xPPFError, tDebouceTimeDoubled := T#300ms, xNoBackupFlag := SYSTEM.stInstrumentFlags.xNoPumpBackup, xRequestPumpSwitch := SYSTEM.stSystemFlags.xSwitchPumpRequest, xAwaitSystemInit := SYSTEM.stSystemFlags.xAwaitInitialization);
SYSTEM.stOutputs.xPump1Activate := fbpumpstartswitchroutine.xPump1ActuationVariable;
SYSTEM.stOutputs.xPump2Activate := fbpumpstartswitchroutine.xPump2ActuationVariable;
xsysalarm4 := fbpumpstartswitchroutine.xSystemAlarm;
xsysfault4 := fbpumpstartswitchroutine.xSystemFault;
(* Network 15 *)
fbtempboundcheck(EN := TRUE, rSystemTemperature := SYSTEM.stInputs.rTemperature, rTempFaultMin := 10, rTempFaultMax := 100, rTempAlarmMin := 30, rTempAlarmMax := 50, tWarningTime := T#100ms, tFailureTime := T#100ms, xAwaitInit := SYSTEM.stSystemFlags.xAwaitInitialization, xAwaitCalibration := SYSTEM.stSystemFlags.xAwaitCalibration, xStartDelay := xStartDelay);
xsysalarm5 := fbtempboundcheck.xTemperatureWarning;
xsysfault5 := fbtempboundcheck.xTemperatureFailure;
(* Network 16 *)
SYSTEM.stSystemFlags.xAlarm := xsysalrm1 OR xsysalarm2 OR xsysalarm3 OR xsysalarm4;
(* Network 17 *)
SYSTEM.stSystemFlags.xFault := xsysfault1 OR xsysfault2 OR xsysfault3 OR xsysfault4;
END_PROGRAM

(* POU System States/FB_InstrumentInputScan, LD *)
FUNCTION_BLOCK FB_InstrumentInputScan
VAR_INPUT
	wPump1Input: WORD;
	wPump2Input: WORD;
	iRTD1Input: INT;
	iRTD2Input: INT;
	iRTD3Input: INT;
	wFlowInput: WORD;
	wConductivityInput: WORD;
	xWaterLowInput: BOOL;
	xWaterLowLowInput: BOOL;
	xConductivityAlarmInput: BOOL;
	xConductivityFaultInput: BOOL;
	xPressureLowInput: BOOL;
	rPump1MaxSignal: REAL;
	rPump2MaxSignal: REAL;
	rRTD1MaxSignal: REAL;
	rRTD2MaxSignal: REAL;
	rRTD3MaxSignal: REAL;
	rFlowMaxSignal: REAL;
	rConductivityMaxSignal: REAL;
	rPump1MinSignal: REAL;
	rPump2MinSignal: REAL;
	rRTD1MinSignal: REAL;
	rRTD2MinSignal: REAL;
	rRTD3MinSignal: REAL;
	rFlowMinSignal: REAL;
	rConductivityMinSignal: REAL;
	rPump1MaxValue: REAL;
	rPump2MaxValue: REAL;
	rRTD1MaxValue: REAL;
	rRTD2MaxValue: REAL;
	rRTD3MaxValue: REAL;
	rFlowMaxValue: REAL;
	rConductivityMaxValue: REAL;
	rPump1MinValue: REAL;
	rPump2MinValue: REAL;
	rRTD1MinValue: REAL;
	rRTD2MinValue: REAL;
	rRTD3MinValue: REAL;
	rFlowMinValue: REAL;
	rConductivityMinValue: REAL;
	rPump1NormTolerance: REAL;
	rPump2NormTolerance: REAL;
	rRTD1NormTolerance: REAL;
	rRTD2NormTolerance: REAL;
	rRTD3NormTolerance: REAL;
	rFlowNormTolerance: REAL;
	rConductivityNormTolerance: REAL;
	tPump1HysteresisTime: TIME;
	tPump2HysteresisTime: TIME;
	tRTD1HysteresisTime: TIME;
	tRTD2HysteresisTime: TIME;
	tRTD3HysteresisTime: TIME;
	tFlowHysteresisTime: TIME;
	tConductivityHysteresisTime: TIME;
	tWaterLowDBTime: TIME;
	tWaterLowLowDBTime: TIME;
	tConductivityAlarmDBTime: TIME;
	tConductivityFaultDBTime: TIME;
	tPressureLowDBTime: TIME;
END_VAR
VAR_OUTPUT
	xPump1BadReadFlag: BOOL;
	xPump2BadReadFlag: BOOL;
	xRTD1BadReadFlag: BOOL;
	xRTD2BadReadFlag: BOOL;
	xRTD3BadReadFlag: BOOL;
	xFlowBadReadFlag: BOOL;
	xConductivityBadReadFlag: BOOL;
	xWaterLowMeasurement: BOOL;
	xWaterLowLowMeasurement: BOOL;
	xConductivityAlarmMeasurement: BOOL;
	xConductivityFaultMeasurement: BOOL;
	xPressureLowMeasurement: BOOL;
END_VAR
VAR
	fbcollectswitchdata: FB_CollectSwitchData;
	fbcollectflowandconductdata: FB_CollectFlowAndConductData;
	fbcollectrtddata: FB_CollectRTDData;
	fbcollectpumpdata: FB_CollectPumpData;
END_VAR
VAR_IN_OUT
	wPump1Signal: WORD;
	wPump2Signal: WORD;
	iRTD1Signal: INT;
	iRTD2Signal: INT;
	iRTD3Signal: INT;
	wFlowSignal: WORD;
	wConductivitySignal: WORD;
	xWaterLowSignal: BOOL;
	xWaterLowLowSignal: BOOL;
	xConductivityAlarmSignal: BOOL;
	xConductivityFaultSignal: BOOL;
	xPressureLowSignal: BOOL;
	rPump1Measurement: REAL;
	rPump2Measurement: REAL;
	rRTD1Measurement: REAL;
	rRTD2Measurement: REAL;
	rRTD3Measurement: REAL;
	rFlowMeasurement: REAL;
	rConductivityMeasurement: REAL;
END_VAR
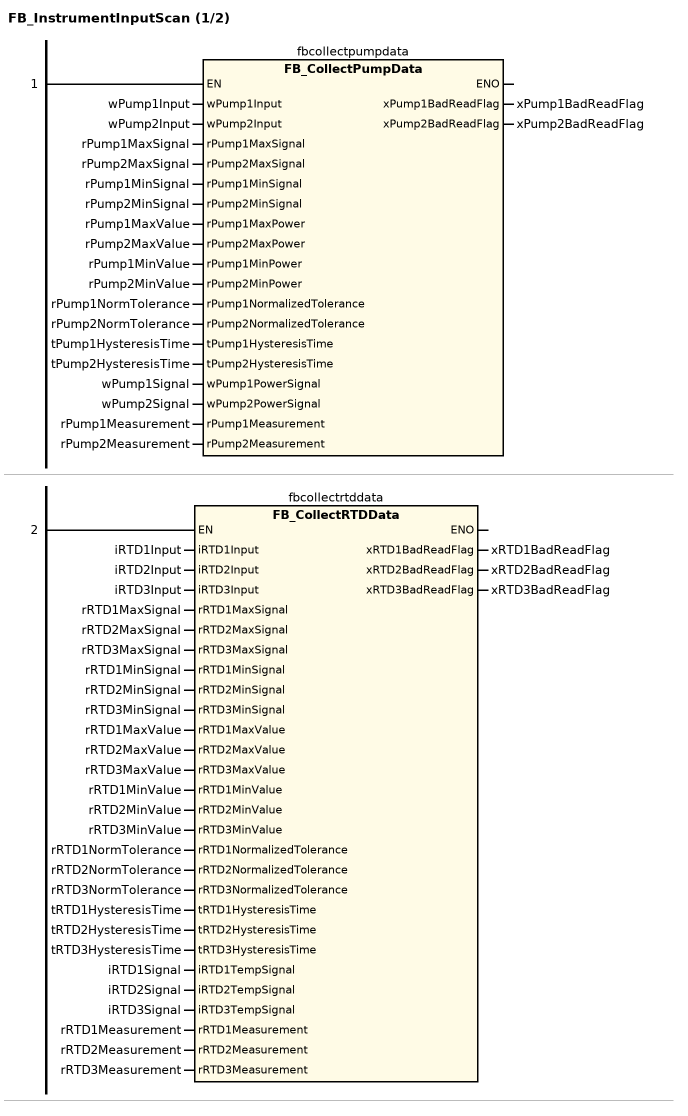
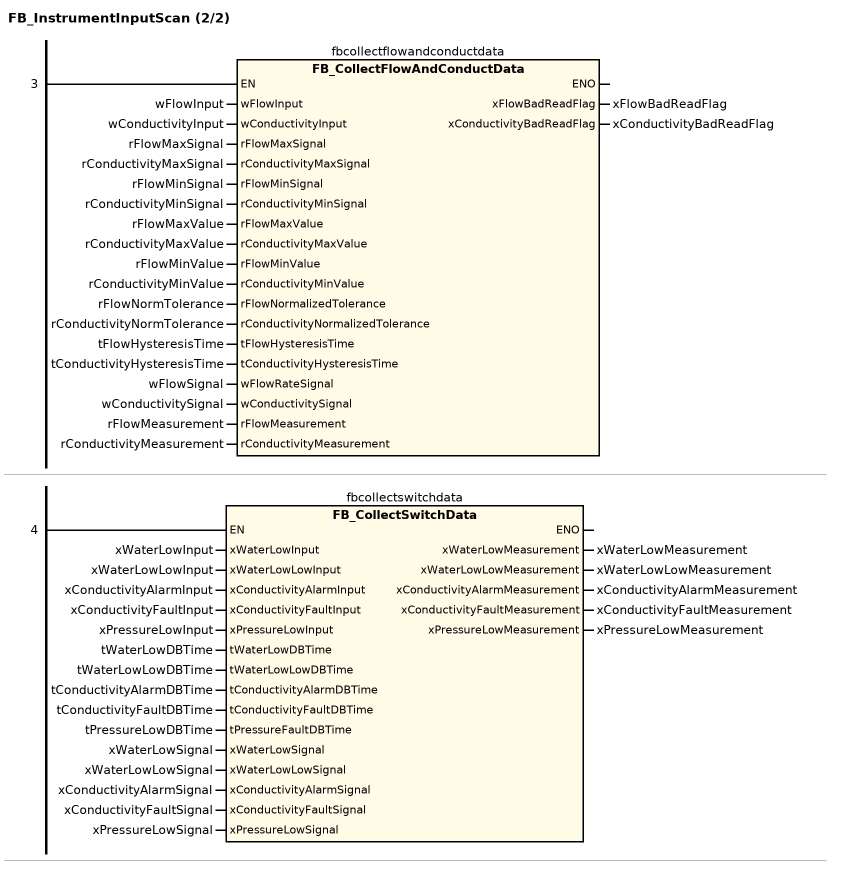
_LD_ (* Ladder Diagram *)
NETWORK 1
	*
		EN --- fbcollectpumpdata:FB_CollectPumpData(wPump1Input: wPump1Input, wPump2Input: wPump2Input, rPump1MaxSignal: rPump1MaxSignal, rPump2MaxSignal: rPump2MaxSignal, rPump1MinSignal: rPump1MinSignal, rPump2MinSignal: rPump2MinSignal, rPump1MaxPower: rPump1MaxValue, rPump2MaxPower: rPump2MaxValue, rPump1MinPower: rPump1MinValue, rPump2MinPower: rPump2MinValue, rPump1NormalizedTolerance: rPump1NormTolerance, rPump2NormalizedTolerance: rPump2NormTolerance, tPump1HysteresisTime: tPump1HysteresisTime, tPump2HysteresisTime: tPump2HysteresisTime, wPump1PowerSignal: wPump1Signal, wPump2PowerSignal: wPump2Signal, rPump1Measurement: rPump1Measurement, rPump2Measurement: rPump2Measurement, xPump2BadReadFlag => xPump2BadReadFlag) => xPump1BadReadFlag
NETWORK 2
	*
		EN --- fbcollectrtddata:FB_CollectRTDData(iRTD1Input: iRTD1Input, iRTD2Input: iRTD2Input, iRTD3Input: iRTD3Input, rRTD1MaxSignal: rRTD1MaxSignal, rRTD2MaxSignal: rRTD2MaxSignal, rRTD3MaxSignal: rRTD3MaxSignal, rRTD1MinSignal: rRTD1MinSignal, rRTD2MinSignal: rRTD2MinSignal, rRTD3MinSignal: rRTD3MinSignal, rRTD1MaxValue: rRTD1MaxValue, rRTD2MaxValue: rRTD2MaxValue, rRTD3MaxValue: rRTD3MaxValue, rRTD1MinValue: rRTD1MinValue, rRTD2MinValue: rRTD2MinValue, rRTD3MinValue: rRTD3MinValue, rRTD1NormalizedTolerance: rRTD1NormTolerance, rRTD2NormalizedTolerance: rRTD2NormTolerance, rRTD3NormalizedTolerance: rRTD3NormTolerance, tRTD1HysteresisTime: tRTD1HysteresisTime, tRTD2HysteresisTime: tRTD2HysteresisTime, tRTD3HysteresisTime: tRTD3HysteresisTime, iRTD1TempSignal: iRTD1Signal, iRTD2TempSignal: iRTD2Signal, iRTD3TempSignal: iRTD3Signal, rRTD1Measurement: rRTD1Measurement, rRTD2Measurement: rRTD2Measurement, rRTD3Measurement: rRTD3Measurement, xRTD2BadReadFlag => xRTD2BadReadFlag, xRTD3BadReadFlag => xRTD3BadReadFlag) => xRTD1BadReadFlag
NETWORK 3
	*
		EN --- fbcollectflowandconductdata:FB_CollectFlowAndConductData(wFlowInput: wFlowInput, wConductivityInput: wConductivityInput, rFlowMaxSignal: rFlowMaxSignal, rConductivityMaxSignal: rConductivityMaxSignal, rFlowMinSignal: rFlowMinSignal, rConductivityMinSignal: rConductivityMinSignal, rFlowMaxValue: rFlowMaxValue, rConductivityMaxValue: rConductivityMaxValue, rFlowMinValue: rFlowMinValue, rConductivityMinValue: rConductivityMinValue, rFlowNormalizedTolerance: rFlowNormTolerance, rConductivityNormalizedTolerance: rConductivityNormTolerance, tFlowHysteresisTime: tFlowHysteresisTime, tConductivityHysteresisTime: tConductivityHysteresisTime, wFlowRateSignal: wFlowSignal, wConductivitySignal: wConductivitySignal, rFlowMeasurement: rFlowMeasurement, rConductivityMeasurement: rConductivityMeasurement, xConductivityBadReadFlag => xConductivityBadReadFlag) => xFlowBadReadFlag
NETWORK 4
	*
		EN --- fbcollectswitchdata:FB_CollectSwitchData(xWaterLowInput: xWaterLowInput, xWaterLowLowInput: xWaterLowLowInput, xConductivityAlarmInput: xConductivityAlarmInput, xConductivityFaultInput: xConductivityFaultInput, xPressureLowInput: xPressureLowInput, tWaterLowDBTime: tWaterLowDBTime, tWaterLowLowDBTime: tWaterLowLowDBTime, tConductivityAlarmDBTime: tConductivityAlarmDBTime, tConductivityFaultDBTime: tConductivityFaultDBTime, tPressureFaultDBTime: tPressureLowDBTime, xWaterLowSignal: xWaterLowSignal, xWaterLowLowSignal: xWaterLowLowSignal, xConductivityAlarmSignal: xConductivityAlarmSignal, xConductivityFaultSignal: xConductivityFaultSignal, xPressureLowSignal: xPressureLowSignal, xWaterLowLowMeasurement => xWaterLowLowMeasurement, xConductivityAlarmMeasurement => xConductivityAlarmMeasurement, xConductivityFaultMeasurement => xConductivityFaultMeasurement, xPressureLowMeasurement => xPressureLowMeasurement) => xWaterLowMeasurement
_END_LD_
(* the same logic as Structured Text *)
(* Network 1 *)
fbcollectpumpdata(wPump1Input := wPump1Input, wPump2Input := wPump2Input, rPump1MaxSignal := rPump1MaxSignal, rPump2MaxSignal := rPump2MaxSignal, rPump1MinSignal := rPump1MinSignal, rPump2MinSignal := rPump2MinSignal, rPump1MaxPower := rPump1MaxValue, rPump2MaxPower := rPump2MaxValue, rPump1MinPower := rPump1MinValue, rPump2MinPower := rPump2MinValue, rPump1NormalizedTolerance := rPump1NormTolerance, rPump2NormalizedTolerance := rPump2NormTolerance, tPump1HysteresisTime := tPump1HysteresisTime, tPump2HysteresisTime := tPump2HysteresisTime, wPump1PowerSignal := wPump1Signal, wPump2PowerSignal := wPump2Signal, rPump1Measurement := rPump1Measurement, rPump2Measurement := rPump2Measurement);
xPump2BadReadFlag := fbcollectpumpdata.xPump2BadReadFlag;
xPump1BadReadFlag := fbcollectpumpdata.xPump1BadReadFlag;
(* Network 2 *)
fbcollectrtddata(iRTD1Input := iRTD1Input, iRTD2Input := iRTD2Input, iRTD3Input := iRTD3Input, rRTD1MaxSignal := rRTD1MaxSignal, rRTD2MaxSignal := rRTD2MaxSignal, rRTD3MaxSignal := rRTD3MaxSignal, rRTD1MinSignal := rRTD1MinSignal, rRTD2MinSignal := rRTD2MinSignal, rRTD3MinSignal := rRTD3MinSignal, rRTD1MaxValue := rRTD1MaxValue, rRTD2MaxValue := rRTD2MaxValue, rRTD3MaxValue := rRTD3MaxValue, rRTD1MinValue := rRTD1MinValue, rRTD2MinValue := rRTD2MinValue, rRTD3MinValue := rRTD3MinValue, rRTD1NormalizedTolerance := rRTD1NormTolerance, rRTD2NormalizedTolerance := rRTD2NormTolerance, rRTD3NormalizedTolerance := rRTD3NormTolerance, tRTD1HysteresisTime := tRTD1HysteresisTime, tRTD2HysteresisTime := tRTD2HysteresisTime, tRTD3HysteresisTime := tRTD3HysteresisTime, iRTD1TempSignal := iRTD1Signal, iRTD2TempSignal := iRTD2Signal, iRTD3TempSignal := iRTD3Signal, rRTD1Measurement := rRTD1Measurement, rRTD2Measurement := rRTD2Measurement, rRTD3Measurement := rRTD3Measurement);
xRTD2BadReadFlag := fbcollectrtddata.xRTD2BadReadFlag;
xRTD3BadReadFlag := fbcollectrtddata.xRTD3BadReadFlag;
xRTD1BadReadFlag := fbcollectrtddata.xRTD1BadReadFlag;
(* Network 3 *)
fbcollectflowandconductdata(wFlowInput := wFlowInput, wConductivityInput := wConductivityInput, rFlowMaxSignal := rFlowMaxSignal, rConductivityMaxSignal := rConductivityMaxSignal, rFlowMinSignal := rFlowMinSignal, rConductivityMinSignal := rConductivityMinSignal, rFlowMaxValue := rFlowMaxValue, rConductivityMaxValue := rConductivityMaxValue, rFlowMinValue := rFlowMinValue, rConductivityMinValue := rConductivityMinValue, rFlowNormalizedTolerance := rFlowNormTolerance, rConductivityNormalizedTolerance := rConductivityNormTolerance, tFlowHysteresisTime := tFlowHysteresisTime, tConductivityHysteresisTime := tConductivityHysteresisTime, wFlowRateSignal := wFlowSignal, wConductivitySignal := wConductivitySignal, rFlowMeasurement := rFlowMeasurement, rConductivityMeasurement := rConductivityMeasurement);
xConductivityBadReadFlag := fbcollectflowandconductdata.xConductivityBadReadFlag;
xFlowBadReadFlag := fbcollectflowandconductdata.xFlowBadReadFlag;
(* Network 4 *)
fbcollectswitchdata(xWaterLowInput := xWaterLowInput, xWaterLowLowInput := xWaterLowLowInput, xConductivityAlarmInput := xConductivityAlarmInput, xConductivityFaultInput := xConductivityFaultInput, xPressureLowInput := xPressureLowInput, tWaterLowDBTime := tWaterLowDBTime, tWaterLowLowDBTime := tWaterLowLowDBTime, tConductivityAlarmDBTime := tConductivityAlarmDBTime, tConductivityFaultDBTime := tConductivityFaultDBTime, tPressureFaultDBTime := tPressureLowDBTime, xWaterLowSignal := xWaterLowSignal, xWaterLowLowSignal := xWaterLowLowSignal, xConductivityAlarmSignal := xConductivityAlarmSignal, xConductivityFaultSignal := xConductivityFaultSignal, xPressureLowSignal := xPressureLowSignal);
xWaterLowLowMeasurement := fbcollectswitchdata.xWaterLowLowMeasurement;
xConductivityAlarmMeasurement := fbcollectswitchdata.xConductivityAlarmMeasurement;
xConductivityFaultMeasurement := fbcollectswitchdata.xConductivityFaultMeasurement;
xPressureLowMeasurement := fbcollectswitchdata.xPressureLowMeasurement;
xWaterLowMeasurement := fbcollectswitchdata.xWaterLowMeasurement;
END_FUNCTION_BLOCK

(* POU System States/FB_CollectSwitchData, LD *)
FUNCTION_BLOCK FB_CollectSwitchData
VAR_INPUT
	xWaterLowInput: BOOL;
	xWaterLowLowInput: BOOL;
	xConductivityAlarmInput: BOOL;
	xConductivityFaultInput: BOOL;
	xPressureLowInput: BOOL;
	tWaterLowDBTime: TIME;
	tWaterLowLowDBTime: TIME;
	tConductivityAlarmDBTime: TIME;
	tConductivityFaultDBTime: TIME;
	tPressureFaultDBTime: TIME;
END_VAR
VAR_OUTPUT
	xWaterLowMeasurement: BOOL;
	xWaterLowLowMeasurement: BOOL;
	xConductivityAlarmMeasurement: BOOL;
	xConductivityFaultMeasurement: BOOL;
	xPressureLowMeasurement: BOOL;
END_VAR
VAR
	fbassigndigitalwaterlow: FB_AssignDigital;
	fbassigndigitalwaterlowlow: FB_AssignDigital;
	fbassigndigitalconductivityalarm: FB_AssignDigital;
	fbassigndigitalconductivityfault: FB_AssignDigital;
	fbassigndigitalpressurelow: FB_AssignDigital;
END_VAR
VAR_IN_OUT
	xWaterLowSignal: BOOL;
	xWaterLowLowSignal: BOOL;
	xConductivityAlarmSignal: BOOL;
	xConductivityFaultSignal: BOOL;
	xPressureLowSignal: BOOL;
END_VAR
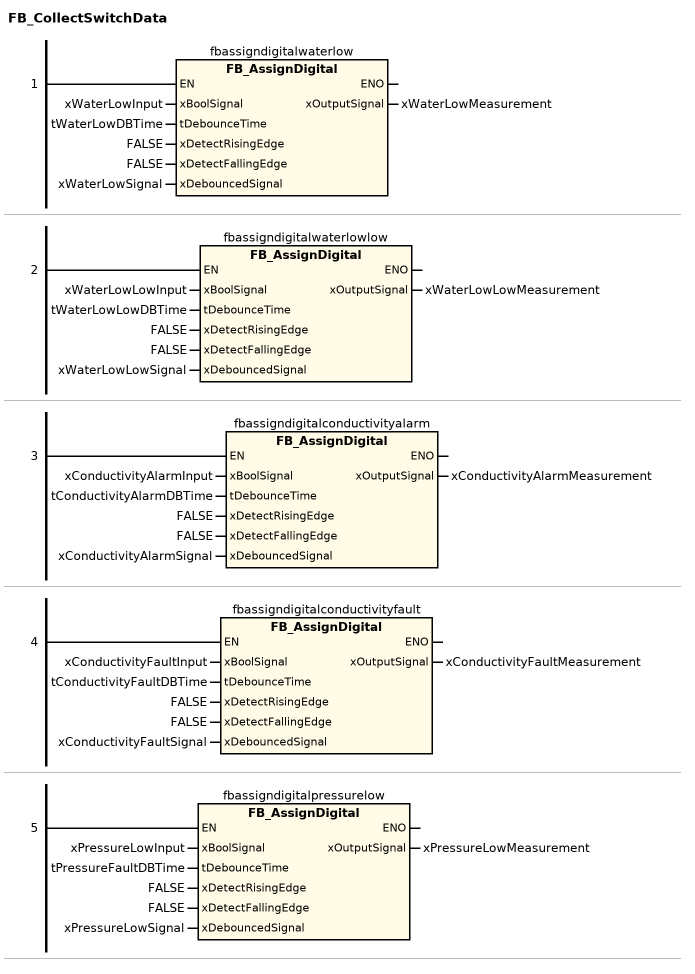
_LD_ (* Ladder Diagram *)
NETWORK 1
	*
		EN --- fbassigndigitalwaterlow:FB_AssignDigital(xBoolSignal: xWaterLowInput, tDebounceTime: tWaterLowDBTime, xDetectRisingEdge: FALSE, xDetectFallingEdge: FALSE, xDebouncedSignal: xWaterLowSignal) => xWaterLowMeasurement
NETWORK 2
	*
		EN --- fbassigndigitalwaterlowlow:FB_AssignDigital(xBoolSignal: xWaterLowLowInput, tDebounceTime: tWaterLowLowDBTime, xDetectRisingEdge: FALSE, xDetectFallingEdge: FALSE, xDebouncedSignal: xWaterLowLowSignal) => xWaterLowLowMeasurement
NETWORK 3
	*
		EN --- fbassigndigitalconductivityalarm:FB_AssignDigital(xBoolSignal: xConductivityAlarmInput, tDebounceTime: tConductivityAlarmDBTime, xDetectRisingEdge: FALSE, xDetectFallingEdge: FALSE, xDebouncedSignal: xConductivityAlarmSignal) => xConductivityAlarmMeasurement
NETWORK 4
	*
		EN --- fbassigndigitalconductivityfault:FB_AssignDigital(xBoolSignal: xConductivityFaultInput, tDebounceTime: tConductivityFaultDBTime, xDetectRisingEdge: FALSE, xDetectFallingEdge: FALSE, xDebouncedSignal: xConductivityFaultSignal) => xConductivityFaultMeasurement
NETWORK 5
	*
		EN --- fbassigndigitalpressurelow:FB_AssignDigital(xBoolSignal: xPressureLowInput, tDebounceTime: tPressureFaultDBTime, xDetectRisingEdge: FALSE, xDetectFallingEdge: FALSE, xDebouncedSignal: xPressureLowSignal) => xPressureLowMeasurement
_END_LD_
(* the same logic as Structured Text *)
(* Network 1 *)
fbassigndigitalwaterlow(xBoolSignal := xWaterLowInput, tDebounceTime := tWaterLowDBTime, xDetectRisingEdge := FALSE, xDetectFallingEdge := FALSE, xDebouncedSignal := xWaterLowSignal);
xWaterLowMeasurement := fbassigndigitalwaterlow.xOutputSignal;
(* Network 2 *)
fbassigndigitalwaterlowlow(xBoolSignal := xWaterLowLowInput, tDebounceTime := tWaterLowLowDBTime, xDetectRisingEdge := FALSE, xDetectFallingEdge := FALSE, xDebouncedSignal := xWaterLowLowSignal);
xWaterLowLowMeasurement := fbassigndigitalwaterlowlow.xOutputSignal;
(* Network 3 *)
fbassigndigitalconductivityalarm(xBoolSignal := xConductivityAlarmInput, tDebounceTime := tConductivityAlarmDBTime, xDetectRisingEdge := FALSE, xDetectFallingEdge := FALSE, xDebouncedSignal := xConductivityAlarmSignal);
xConductivityAlarmMeasurement := fbassigndigitalconductivityalarm.xOutputSignal;
(* Network 4 *)
fbassigndigitalconductivityfault(xBoolSignal := xConductivityFaultInput, tDebounceTime := tConductivityFaultDBTime, xDetectRisingEdge := FALSE, xDetectFallingEdge := FALSE, xDebouncedSignal := xConductivityFaultSignal);
xConductivityFaultMeasurement := fbassigndigitalconductivityfault.xOutputSignal;
(* Network 5 *)
fbassigndigitalpressurelow(xBoolSignal := xPressureLowInput, tDebounceTime := tPressureFaultDBTime, xDetectRisingEdge := FALSE, xDetectFallingEdge := FALSE, xDebouncedSignal := xPressureLowSignal);
xPressureLowMeasurement := fbassigndigitalpressurelow.xOutputSignal;
END_FUNCTION_BLOCK

(* POU Data Conversion/Signal->Instrument/FB_AssignDigital, LD *)
FUNCTION_BLOCK FB_AssignDigital
VAR_INPUT
	xBoolSignal: BOOL;
	tDebounceTime: TIME;
	xDetectRisingEdge: BOOL;
	xDetectFallingEdge: BOOL;
END_VAR
VAR_OUTPUT
	xOutputSignal: BOOL;
END_VAR
VAR

	fbRise: R_TRIG;
	fbRTrig: R_TRIG;
	xSignalRise: BOOL;
	fbFTrig: F_TRIG;
	xSignalFall: BOOL;
	xEdgeSignal1: BOOL;
	xEdgeSignal: BOOL;
	fbdesig: FB_DebounceSignal;
END_VAR
VAR_IN_OUT
	xDebouncedSignal: BOOL;
END_VAR
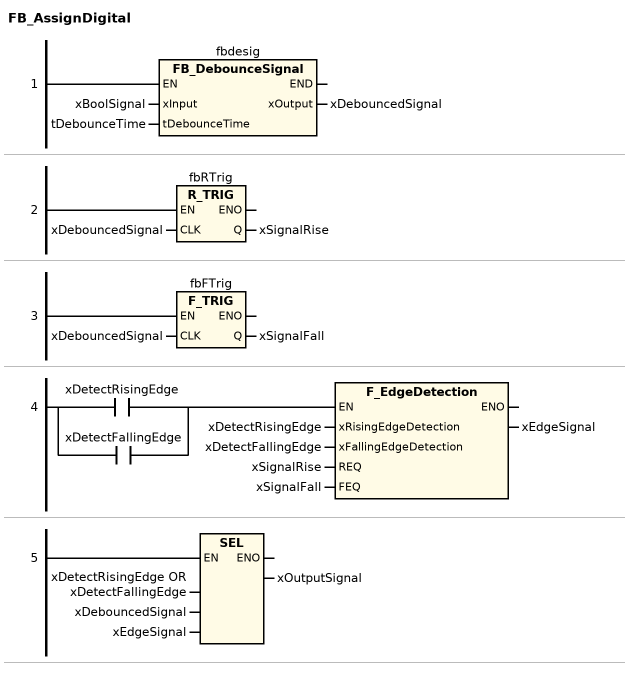
_LD_ (* Ladder Diagram *)
NETWORK 1
	fbdesig:FB_DebounceSignal(EN: *, xInput: xBoolSignal, tDebounceTime: tDebounceTime, xOutput => xDebouncedSignal)
NETWORK 2
	*
		EN --- fbRTrig:R_TRIG(CLK: xDebouncedSignal) => xSignalRise
NETWORK 3
	*
		EN --- fbFTrig:F_TRIG(CLK: xDebouncedSignal) => xSignalFall
NETWORK 4
	{ [xDetectRisingEdge] | [xDetectFallingEdge] }
		EN --- F_EdgeDetection(xRisingEdgeDetection: xDetectRisingEdge, xFallingEdgeDetection: xDetectFallingEdge, REQ: xSignalRise, FEQ: xSignalFall) => xEdgeSignal
NETWORK 5
	*
		EN --- SEL(xDetectRisingEdge OR xDetectFallingEdge, xDebouncedSignal, xEdgeSignal) => xOutputSignal
_END_LD_
(* the same logic as Structured Text *)
(* Network 1 *)
fbdesig(EN := TRUE, xInput := xBoolSignal, tDebounceTime := tDebounceTime);
xDebouncedSignal := fbdesig.xOutput;
(* Network 2 *)
fbRTrig(CLK := xDebouncedSignal);
xSignalRise := fbRTrig.Q;
(* Network 3 *)
fbFTrig(CLK := xDebouncedSignal);
xSignalFall := fbFTrig.Q;
(* Network 4 *)
IF xDetectRisingEdge OR xDetectFallingEdge THEN
	xEdgeSignal := F_EdgeDetection(xRisingEdgeDetection := xDetectRisingEdge, xFallingEdgeDetection := xDetectFallingEdge, REQ := xSignalRise, FEQ := xSignalFall);
END_IF;
(* Network 5 *)
xOutputSignal := SEL(xDetectRisingEdge OR xDetectFallingEdge, xDebouncedSignal, xEdgeSignal);
END_FUNCTION_BLOCK

(* POU Functions/FB_DebounceSignal, ST *)
FUNCTION_BLOCK FB_DebounceSignal
VAR_INPUT
	EN: BOOL;
	xInput: BOOL;
	tDebounceTime: TIME;
END_VAR
VAR_OUTPUT
	END: BOOL;
	xOutput: BOOL;
END_VAR
VAR
	fbDebounceTimerON: TON;
	fbDebounceTimerOFF: TOF;
END_VAR
IF EN  = FALSE THEN
	RETURN;
END_IF

fbDebounceTimerON(IN := xInput, PT := tDebounceTime); (*Won't go to true until 50 ms of stability. Every false resets this timer*)

fbDebounceTimerOFF(IN := fbDebounceTimerON.Q, PT := tDebounceTime); (*Won't go to false until 50ms of stability. Every true resets this timer*)
xOutput  := fbDebounceTimerOFF.Q;

END := TRUE;
END_FUNCTION_BLOCK

(* POU Functions/F_EdgeDetection, ST *)
FUNCTION F_EdgeDetection : BOOL
VAR_INPUT
	xRisingEdgeDetection: BOOL;
	xFallingEdgeDetection: BOOL;
	REQ: BOOL;
	FEQ: BOOL;
END_VAR
VAR
END_VAR
IF xRisingEdgeDetection = TRUE AND xFallingEdgeDetection = TRUE THEN
	F_EdgeDetection := REQ OR FEQ; (*Are we detecing if this goes from False to True. When we detect this, caputre it*)
ELSIF xFallingEdgeDetection = TRUE THEN
	F_EdgeDetection := FEQ; (*Same as above but Vice Versa. Note that you can have both!*)
ELSIF xRisingEdgeDetection = TRUE THEN
	F_EdgeDetection  := REQ;
END_IF
END_FUNCTION

(* POU System States/FB_CollectFlowAndConductData, LD *)
FUNCTION_BLOCK FB_CollectFlowAndConductData
VAR_INPUT
	wFlowInput: WORD;
	wConductivityInput: WORD;
	rFlowMaxSignal: REAL;
	rConductivityMaxSignal: REAL;
	rFlowMinSignal: REAL;
	rConductivityMinSignal: REAL;
	rFlowMaxValue: REAL;
	rConductivityMaxValue: REAL;
	rFlowMinValue: REAL;
	rConductivityMinValue: REAL;
	rFlowNormalizedTolerance: REAL;
	rConductivityNormalizedTolerance: REAL;
	tFlowHysteresisTime: TIME;
	tConductivityHysteresisTime: TIME;
END_VAR
VAR_OUTPUT
	xFlowBadReadFlag: BOOL;
	xConductivityBadReadFlag: BOOL;
END_VAR
VAR
	fbassignanalogflow: FB_AssignAnalog;
	fbassignanalogconductivity: FB_AssignAnalog;
	emptyi: INT;
END_VAR
VAR CONSTANT

END_VAR
VAR CONSTANT
END_VAR
VAR_IN_OUT
	wFlowRateSignal: WORD;
	wConductivitySignal: WORD;
	rFlowMeasurement: REAL;
	rConductivityMeasurement: REAL;
END_VAR
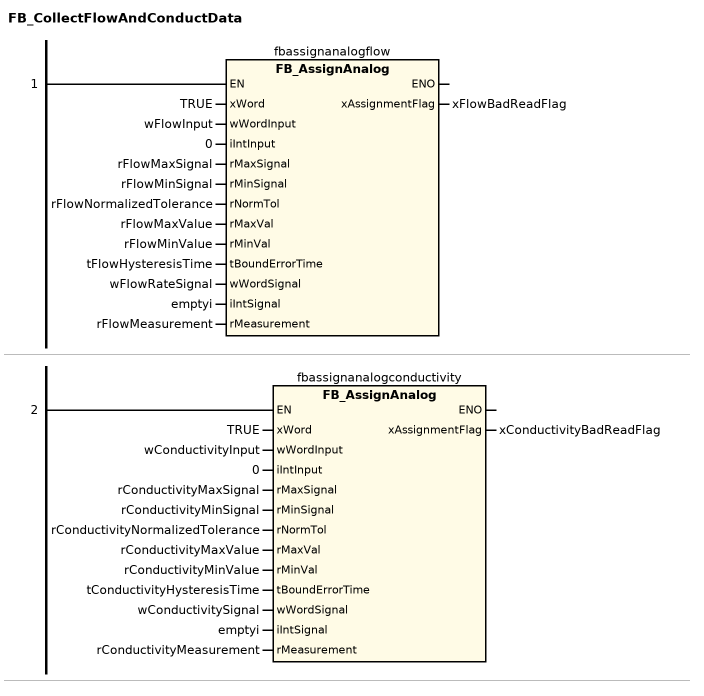
_LD_ (* Ladder Diagram *)
NETWORK 1
	*
		EN --- fbassignanalogflow:FB_AssignAnalog(xWord: TRUE, wWordInput: wFlowInput, iIntInput: 0, rMaxSignal: rFlowMaxSignal, rMinSignal: rFlowMinSignal, rNormTol: rFlowNormalizedTolerance, rMaxVal: rFlowMaxValue, rMinVal: rFlowMinValue, tBoundErrorTime: tFlowHysteresisTime, wWordSignal: wFlowRateSignal, iIntSignal: emptyi, rMeasurement: rFlowMeasurement) => xFlowBadReadFlag
NETWORK 2
	*
		EN --- fbassignanalogconductivity:FB_AssignAnalog(xWord: TRUE, wWordInput: wConductivityInput, iIntInput: 0, rMaxSignal: rConductivityMaxSignal, rMinSignal: rConductivityMinSignal, rNormTol: rConductivityNormalizedTolerance, rMaxVal: rConductivityMaxValue, rMinVal: rConductivityMinValue, tBoundErrorTime: tConductivityHysteresisTime, wWordSignal: wConductivitySignal, iIntSignal: emptyi, rMeasurement: rConductivityMeasurement) => xConductivityBadReadFlag
_END_LD_
(* the same logic as Structured Text *)
(* Network 1 *)
fbassignanalogflow(xWord := TRUE, wWordInput := wFlowInput, iIntInput := 0, rMaxSignal := rFlowMaxSignal, rMinSignal := rFlowMinSignal, rNormTol := rFlowNormalizedTolerance, rMaxVal := rFlowMaxValue, rMinVal := rFlowMinValue, tBoundErrorTime := tFlowHysteresisTime, wWordSignal := wFlowRateSignal, iIntSignal := emptyi, rMeasurement := rFlowMeasurement);
xFlowBadReadFlag := fbassignanalogflow.xAssignmentFlag;
(* Network 2 *)
fbassignanalogconductivity(xWord := TRUE, wWordInput := wConductivityInput, iIntInput := 0, rMaxSignal := rConductivityMaxSignal, rMinSignal := rConductivityMinSignal, rNormTol := rConductivityNormalizedTolerance, rMaxVal := rConductivityMaxValue, rMinVal := rConductivityMinValue, tBoundErrorTime := tConductivityHysteresisTime, wWordSignal := wConductivitySignal, iIntSignal := emptyi, rMeasurement := rConductivityMeasurement);
xConductivityBadReadFlag := fbassignanalogconductivity.xAssignmentFlag;
END_FUNCTION_BLOCK

(* POU Data Conversion/Signal->Instrument/FB_AssignAnalog, LD *)
FUNCTION_BLOCK FB_AssignAnalog
VAR_INPUT
	xWord: BOOL;
	wWordInput: WORD;
	iIntInput: INT;
	rMaxSignal: REAL;
	rMinSignal: REAL;
	rNormTol: REAL;
	rMaxVal: REAL;
	rMinVal: REAL;
	tBoundErrorTime: TIME;
END_VAR
VAR_OUTPUT
	xAssignmentFlag: BOOL;

END_VAR
VAR
	rSignal: REAL;
	rNormalizedSignal: REAL;
		rSignal1: REAL;
		rSignal2: REAL;
		rLastRead: REAL;
		rLinearizedSignal: REAL;
		xBoundError: BOOL;
		fbTON: TON;
		fbvalcap: FB_ValueCap;
	fbdebounce: FB_DebounceSignal;
END_VAR

VAR_IN_OUT
	wWordSignal: WORD;
	iIntSignal: INT;
	rMeasurement: REAL;
END_VAR
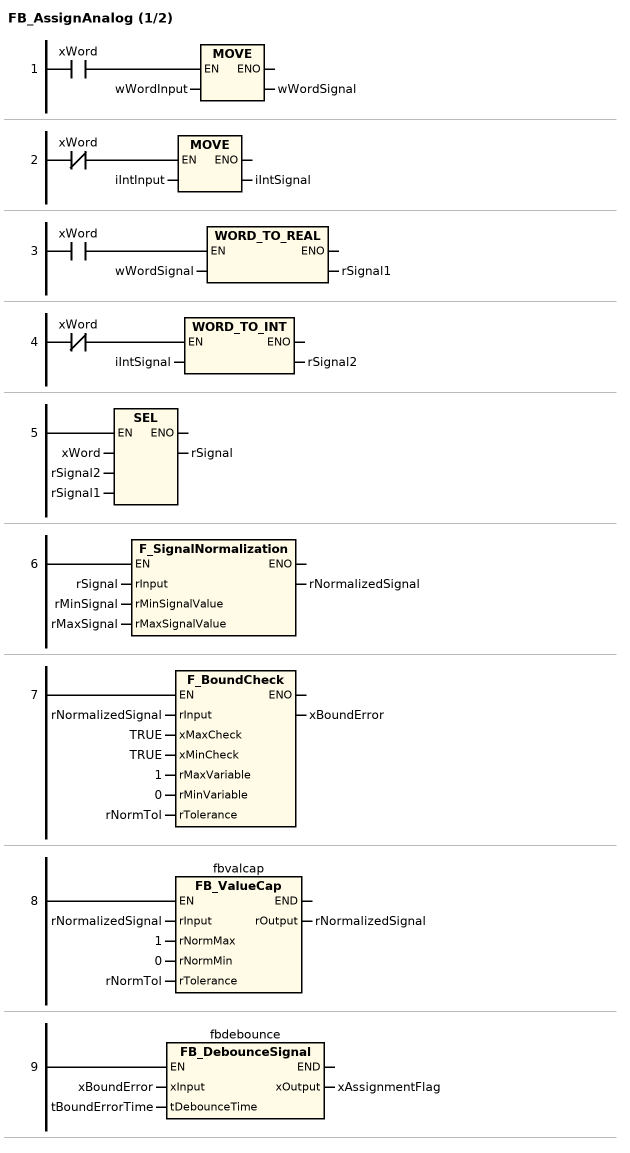
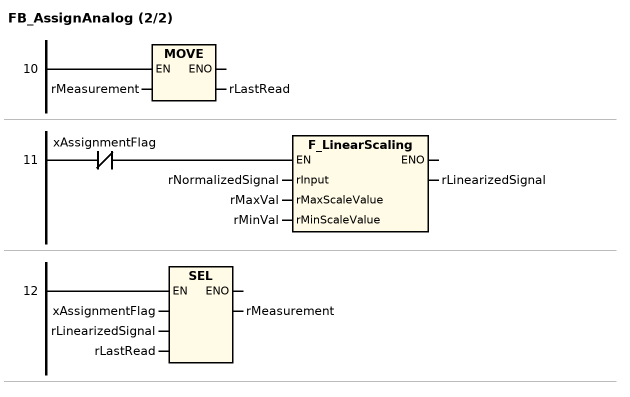
_LD_ (* Ladder Diagram *)
NETWORK 1
	[xWord]
		EN --- MOVE(wWordInput) => wWordSignal
NETWORK 2
	[/xWord]
		EN --- MOVE(iIntInput) => iIntSignal
NETWORK 3
	[xWord]
		EN --- WORD_TO_REAL(wWordSignal) => rSignal1
NETWORK 4
	[/xWord]
		EN --- WORD_TO_INT(iIntSignal) => rSignal2
NETWORK 5
	*
		EN --- SEL(xWord, rSignal2, rSignal1) => rSignal
NETWORK 6
	*
		EN --- F_SignalNormalization(rInput: rSignal, rMinSignalValue: rMinSignal, rMaxSignalValue: rMaxSignal) => rNormalizedSignal
NETWORK 7
	*
		EN --- F_BoundCheck(rInput: rNormalizedSignal, xMaxCheck: TRUE, xMinCheck: TRUE, rMaxVariable: 1, rMinVariable: 0, rTolerance: rNormTol) => xBoundError
NETWORK 8
	fbvalcap:FB_ValueCap(EN: *, rInput: rNormalizedSignal, rNormMax: 1, rNormMin: 0, rTolerance: rNormTol, rOutput => rNormalizedSignal)
NETWORK 9
	fbdebounce:FB_DebounceSignal(EN: *, xInput: xBoundError, tDebounceTime: tBoundErrorTime, xOutput => xAssignmentFlag)
NETWORK 10
	*
		EN --- MOVE(rMeasurement) => rLastRead
NETWORK 11
	[/xAssignmentFlag]
		EN --- F_LinearScaling(rInput: rNormalizedSignal, rMaxScaleValue: rMaxVal, rMinScaleValue: rMinVal) => rLinearizedSignal
NETWORK 12
	*
		EN --- SEL(xAssignmentFlag, rLinearizedSignal, rLastRead) => rMeasurement
_END_LD_
(* the same logic as Structured Text *)
(* Network 1 *)
IF xWord THEN
	wWordSignal := wWordInput;
END_IF;
(* Network 2 *)
IF NOT xWord THEN
	iIntSignal := iIntInput;
END_IF;
(* Network 3 *)
IF xWord THEN
	rSignal1 := WORD_TO_REAL(wWordSignal);
END_IF;
(* Network 4 *)
IF NOT xWord THEN
	rSignal2 := WORD_TO_INT(iIntSignal);
END_IF;
(* Network 5 *)
rSignal := SEL(xWord, rSignal2, rSignal1);
(* Network 6 *)
rNormalizedSignal := F_SignalNormalization(rInput := rSignal, rMinSignalValue := rMinSignal, rMaxSignalValue := rMaxSignal);
(* Network 7 *)
xBoundError := F_BoundCheck(rInput := rNormalizedSignal, xMaxCheck := TRUE, xMinCheck := TRUE, rMaxVariable := 1, rMinVariable := 0, rTolerance := rNormTol);
(* Network 8 *)
fbvalcap(EN := TRUE, rInput := rNormalizedSignal, rNormMax := 1, rNormMin := 0, rTolerance := rNormTol);
rNormalizedSignal := fbvalcap.rOutput;
(* Network 9 *)
fbdebounce(EN := TRUE, xInput := xBoundError, tDebounceTime := tBoundErrorTime);
xAssignmentFlag := fbdebounce.xOutput;
(* Network 10 *)
rLastRead := rMeasurement;
(* Network 11 *)
IF NOT xAssignmentFlag THEN
	rLinearizedSignal := F_LinearScaling(rInput := rNormalizedSignal, rMaxScaleValue := rMaxVal, rMinScaleValue := rMinVal);
END_IF;
(* Network 12 *)
rMeasurement := SEL(xAssignmentFlag, rLinearizedSignal, rLastRead);
END_FUNCTION_BLOCK

(* POU Functions/FB_ValueCap, ST *)
FUNCTION_BLOCK FB_ValueCap
VAR_INPUT
	EN: BOOL;
	rInput: REAL;
	rNormMax: REAL;
	rNormMin: REAL;
	rTolerance: REAL;
END_VAR
VAR_OUTPUT
	END: BOOL;
	rOutput: REAL;
END_VAR
VAR
	rLastRead: REAL := 0;
END_VAR
IF (rInput > rNormMax + rTolerance) OR (rInput < rNormMin - rTolerance) THEN
	rOutput  := rLastRead;
ELSIF (rInput > 1) THEN
	rOutput := 1;
	rLastRead := 1;
ELSIF (rInput < 0) THEN
	rOutput := 0;
	rLastRead := 0;
ELSE
	rOutput := rInput;
	rLastRead := rInput;
END_IF
END_FUNCTION_BLOCK

(* POU Functions/F_SignalNormalization, ST *)
FUNCTION F_SignalNormalization : REAL
VAR_INPUT
	rInput: REAL;
	rMinSignalValue: REAL;
	rMaxSignalValue: REAL;
END_VAR
VAR
END_VAR
IF rMinSignalValue > rMaxSignalValue OR rMinSignalValue = rMaxSignalValue THEN
	F_SignalNormalization := 0;
ELSE
	F_SignalNormalization  := ((rInput - rMinSignalValue)) / (rMaxSignalValue - rMinSignalValue);
END_IF
;
END_FUNCTION

(* POU Instrument Checking Functions/F_BoundCheck, ST *)
FUNCTION F_BoundCheck : BOOL
VAR_INPUT
	rInput: REAL;
	xMaxCheck: BOOL;
	xMinCheck: BOOL;
	rMaxVariable: REAL;
	rMinVariable: REAL;
	rTolerance: REAL;
END_VAR
VAR
	xPastBoundFlag: BOOL;
END_VAR
xPastBoundFlag := FALSE;
IF xMaxCheck = TRUE AND xMinCheck = TRUE THEN
	IF rInput > (rMaxVariable + rTolerance) THEN
		xPastBoundFlag := TRUE;
	ELSIF rInput < (rMinVariable - rTolerance) THEN
		xPastBoundFlag := TRUE;
	END_IF
ELSIF xMaxCheck = TRUE THEN
	IF rInput > (rMaxVariable + rTolerance) THEN
		xPastBoundFlag := TRUE;
	END_IF
ELSIF xMinCheck = TRUE THEN
	IF rInput < (rMinVariable - rTolerance) THEN
		xPastBoundFlag := TRUE;
	END_IF
END_IF

F_BoundCheck := xPastBoundFlag;
END_FUNCTION

(* POU Functions/F_LinearScaling, ST *)
FUNCTION F_LinearScaling : REAL
VAR_INPUT
	rInput: REAL;
	rMaxScaleValue: REAL;
	rMinScaleValue: REAL;
END_VAR
VAR
END_VAR
IF rMaxScaleValue <  rMinScaleValue OR rMaxScaleValue = rMinScaleValue THEN
	F_LinearScaling := 0;
ELSE
	F_LinearScaling := rInput * (rMaxScaleValue - rMinScaleValue) + rMinScaleValue;
END_IF
END_FUNCTION

(* POU System States/FB_CollectRTDData, LD *)
FUNCTION_BLOCK FB_CollectRTDData
VAR_INPUT
	iRTD1Input: INT;
	iRTD2Input: INT;
	iRTD3Input: INT;
	rRTD1MaxSignal: REAL;
	rRTD2MaxSignal: REAL;
	rRTD3MaxSignal: REAL;
	rRTD1MinSignal: REAL;
	rRTD2MinSignal: REAL;
	rRTD3MinSignal: REAL;
	rRTD1MaxValue: REAL;
	rRTD2MaxValue: REAL;
	rRTD3MaxValue: REAL;
	rRTD1MinValue: REAL;
	rRTD2MinValue: REAL;
	rRTD3MinValue: REAL;
	rRTD1NormalizedTolerance: REAL;
	rRTD2NormalizedTolerance: REAL;
	rRTD3NormalizedTolerance: REAL;
	tRTD1HysteresisTime: TIME;
	tRTD2HysteresisTime: TIME;
	tRTD3HysteresisTime: TIME;
END_VAR
VAR_OUTPUT
	xRTD1BadReadFlag: BOOL;
	xRTD2BadReadFlag: BOOL;
	xRTD3BadReadFlag: BOOL;
END_VAR
VAR
	fbassignanalogRTD1: FB_AssignAnalog;
	fbassignanalogRTD2: FB_AssignAnalog;
	fbassignanalogRTD3: FB_AssignAnalog;
	emptyword: WORD;
END_VAR
VAR CONSTANT

END_VAR
VAR CONSTANT
END_VAR
VAR_IN_OUT
	iRTD1TempSignal: INT;
	iRTD2TempSignal: INT;
	iRTD3TempSignal: INT;
	rRTD1Measurement: REAL;
	rRTD2Measurement: REAL;
	rRTD3Measurement: REAL;
END_VAR
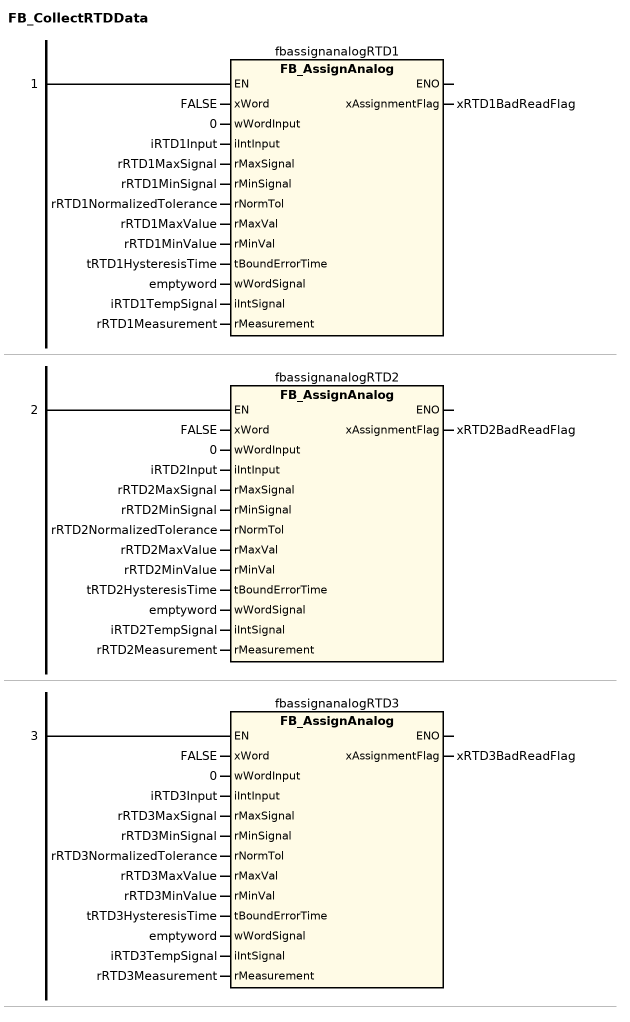
_LD_ (* Ladder Diagram *)
NETWORK 1
	*
		EN --- fbassignanalogRTD1:FB_AssignAnalog(xWord: FALSE, wWordInput: 0, iIntInput: iRTD1Input, rMaxSignal: rRTD1MaxSignal, rMinSignal: rRTD1MinSignal, rNormTol: rRTD1NormalizedTolerance, rMaxVal: rRTD1MaxValue, rMinVal: rRTD1MinValue, tBoundErrorTime: tRTD1HysteresisTime, wWordSignal: emptyword, iIntSignal: iRTD1TempSignal, rMeasurement: rRTD1Measurement) => xRTD1BadReadFlag
NETWORK 2
	*
		EN --- fbassignanalogRTD2:FB_AssignAnalog(xWord: FALSE, wWordInput: 0, iIntInput: iRTD2Input, rMaxSignal: rRTD2MaxSignal, rMinSignal: rRTD2MinSignal, rNormTol: rRTD2NormalizedTolerance, rMaxVal: rRTD2MaxValue, rMinVal: rRTD2MinValue, tBoundErrorTime: tRTD2HysteresisTime, wWordSignal: emptyword, iIntSignal: iRTD2TempSignal, rMeasurement: rRTD2Measurement) => xRTD2BadReadFlag
NETWORK 3
	*
		EN --- fbassignanalogRTD3:FB_AssignAnalog(xWord: FALSE, wWordInput: 0, iIntInput: iRTD3Input, rMaxSignal: rRTD3MaxSignal, rMinSignal: rRTD3MinSignal, rNormTol: rRTD3NormalizedTolerance, rMaxVal: rRTD3MaxValue, rMinVal: rRTD3MinValue, tBoundErrorTime: tRTD3HysteresisTime, wWordSignal: emptyword, iIntSignal: iRTD3TempSignal, rMeasurement: rRTD3Measurement) => xRTD3BadReadFlag
_END_LD_
(* the same logic as Structured Text *)
(* Network 1 *)
fbassignanalogRTD1(xWord := FALSE, wWordInput := 0, iIntInput := iRTD1Input, rMaxSignal := rRTD1MaxSignal, rMinSignal := rRTD1MinSignal, rNormTol := rRTD1NormalizedTolerance, rMaxVal := rRTD1MaxValue, rMinVal := rRTD1MinValue, tBoundErrorTime := tRTD1HysteresisTime, wWordSignal := emptyword, iIntSignal := iRTD1TempSignal, rMeasurement := rRTD1Measurement);
xRTD1BadReadFlag := fbassignanalogRTD1.xAssignmentFlag;
(* Network 2 *)
fbassignanalogRTD2(xWord := FALSE, wWordInput := 0, iIntInput := iRTD2Input, rMaxSignal := rRTD2MaxSignal, rMinSignal := rRTD2MinSignal, rNormTol := rRTD2NormalizedTolerance, rMaxVal := rRTD2MaxValue, rMinVal := rRTD2MinValue, tBoundErrorTime := tRTD2HysteresisTime, wWordSignal := emptyword, iIntSignal := iRTD2TempSignal, rMeasurement := rRTD2Measurement);
xRTD2BadReadFlag := fbassignanalogRTD2.xAssignmentFlag;
(* Network 3 *)
fbassignanalogRTD3(xWord := FALSE, wWordInput := 0, iIntInput := iRTD3Input, rMaxSignal := rRTD3MaxSignal, rMinSignal := rRTD3MinSignal, rNormTol := rRTD3NormalizedTolerance, rMaxVal := rRTD3MaxValue, rMinVal := rRTD3MinValue, tBoundErrorTime := tRTD3HysteresisTime, wWordSignal := emptyword, iIntSignal := iRTD3TempSignal, rMeasurement := rRTD3Measurement);
xRTD3BadReadFlag := fbassignanalogRTD3.xAssignmentFlag;
END_FUNCTION_BLOCK

(* POU System States/FB_CollectPumpData, LD *)
FUNCTION_BLOCK FB_CollectPumpData
VAR_INPUT
	wPump1Input: WORD;
	wPump2Input: WORD;
	rPump1MaxSignal: REAL;
	rPump2MaxSignal: REAL;
	rPump1MinSignal: REAL;
	rPump2MinSignal: REAL;
	rPump1MaxPower: REAL;
	rPump2MaxPower: REAL;
	rPump1MinPower: REAL;
	rPump2MinPower: REAL;
	rPump1NormalizedTolerance: REAL;
	rPump2NormalizedTolerance: REAL;
	tPump1HysteresisTime: TIME;
	tPump2HysteresisTime: TIME;
END_VAR
VAR_OUTPUT
	xPump1BadReadFlag: BOOL;
	xPump2BadReadFlag: BOOL;
END_VAR
VAR
	fbassignanalogpump1: FB_AssignAnalog;
	fbassignanalogpump2: FB_AssignAnalog;
	emptyi: INT;
END_VAR
VAR CONSTANT

END_VAR
VAR CONSTANT
END_VAR
VAR_IN_OUT
	wPump1PowerSignal: WORD;
	wPump2PowerSignal: WORD;
	rPump1Measurement: REAL;
	rPump2Measurement: REAL;
END_VAR
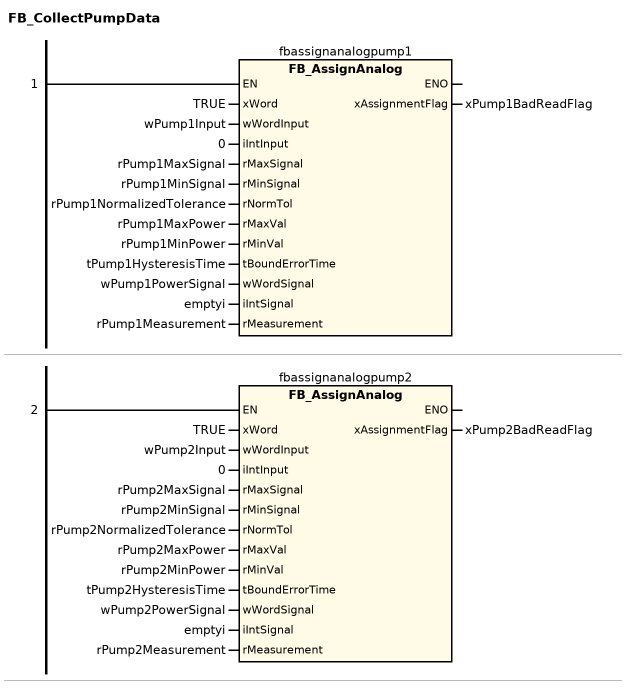
_LD_ (* Ladder Diagram *)
NETWORK 1
	*
		EN --- fbassignanalogpump1:FB_AssignAnalog(xWord: TRUE, wWordInput: wPump1Input, iIntInput: 0, rMaxSignal: rPump1MaxSignal, rMinSignal: rPump1MinSignal, rNormTol: rPump1NormalizedTolerance, rMaxVal: rPump1MaxPower, rMinVal: rPump1MinPower, tBoundErrorTime: tPump1HysteresisTime, wWordSignal: wPump1PowerSignal, iIntSignal: emptyi, rMeasurement: rPump1Measurement) => xPump1BadReadFlag
NETWORK 2
	*
		EN --- fbassignanalogpump2:FB_AssignAnalog(xWord: TRUE, wWordInput: wPump2Input, iIntInput: 0, rMaxSignal: rPump2MaxSignal, rMinSignal: rPump2MinSignal, rNormTol: rPump2NormalizedTolerance, rMaxVal: rPump2MaxPower, rMinVal: rPump2MinPower, tBoundErrorTime: tPump2HysteresisTime, wWordSignal: wPump2PowerSignal, iIntSignal: emptyi, rMeasurement: rPump2Measurement) => xPump2BadReadFlag
_END_LD_
(* the same logic as Structured Text *)
(* Network 1 *)
fbassignanalogpump1(xWord := TRUE, wWordInput := wPump1Input, iIntInput := 0, rMaxSignal := rPump1MaxSignal, rMinSignal := rPump1MinSignal, rNormTol := rPump1NormalizedTolerance, rMaxVal := rPump1MaxPower, rMinVal := rPump1MinPower, tBoundErrorTime := tPump1HysteresisTime, wWordSignal := wPump1PowerSignal, iIntSignal := emptyi, rMeasurement := rPump1Measurement);
xPump1BadReadFlag := fbassignanalogpump1.xAssignmentFlag;
(* Network 2 *)
fbassignanalogpump2(xWord := TRUE, wWordInput := wPump2Input, iIntInput := 0, rMaxSignal := rPump2MaxSignal, rMinSignal := rPump2MinSignal, rNormTol := rPump2NormalizedTolerance, rMaxVal := rPump2MaxPower, rMinVal := rPump2MinPower, tBoundErrorTime := tPump2HysteresisTime, wWordSignal := wPump2PowerSignal, iIntSignal := emptyi, rMeasurement := rPump2Measurement);
xPump2BadReadFlag := fbassignanalogpump2.xAssignmentFlag;
END_FUNCTION_BLOCK

(* POU Data Conversion/Instrument->System/FB_SystemInstrumentAlignment, LD *)
FUNCTION_BLOCK FB_SystemInstrumentAlignment
VAR_INPUT
	EN: BOOL;
	xPump1Fault: BOOL;
	xPump2Fault: BOOL;
	xConductivitySensorError: BOOL;
	xFlowSensorError: BOOL;
	xPressureLowSwtich: BOOL;
	xWaterLevelLowSwtich: BOOL;
	xWaterLevelLowLowSwtich: BOOL;
	xConductivityAlarmSwitch: BOOL;
	xConductivityFaultSwitch: BOOL;
	rConduvitySensorMeasurement: REAL;
	rFlowSensorMeasurement: REAL;
	iActivePump: INT;
	rPump1Power: REAL;
	rPump2Power: REAL;
	rTemp1: REAL;
	rTemp2: REAL;
	rTemp3: REAL;
	xTemp1Flag: BOOL;
	xTemp2Flag: BOOL;
	xTemp3Flag: BOOL;

END_VAR
VAR_OUTPUT
	END: BOOL;
	xSystemAlarmFlag: BOOL;
	xSystemFaultFlag: BOOL;
	rSystemConductivityMeasurement: REAL;
	rSystemFlowMeasurement: REAL;
	rSystemPumpPower: REAL;
	xRequestPumpSwitch: BOOL;
	iPumpFaultCount: INT;
	rSystemMeasuredTemp: REAL;
	iRTDFaultCount: INT;
	xSystemPressureLow: BOOL;
	xSystemWaterLevelLow: BOOL;
	xSystemWaterLevelLowLow: BOOL;
	xSystemConductivityAlarm: BOOL;
	xSystemConductivityFault: BOOL;

END_VAR
VAR
	fbcfsa: FB_CondFlowSystemAlignment;
	fbcfsa2: FB_CondFlowSystemAlignment;
	fbpsa: FB_PumpSystemAlignment;

	fbtsa: FB_TempSystemAlignment;

	xSystemFaultFlag1: BOOL;
	xSystemFaultFlag2: BOOL;
	xSystemFaultFlag3: BOOL;
	xSystemFaultFlag4: BOOL;
	xSystemAlarmFlag1: BOOL;
	xSystemAlarmFlag2: BOOL;
	xSystemAlarmFlag3: BOOL;
	xSAFcontact: BOOL;
	xSAAcontact: BOOL;
END_VAR
VAR_IN_OUT
	xNoBackupFlag: BOOL;

END_VAR
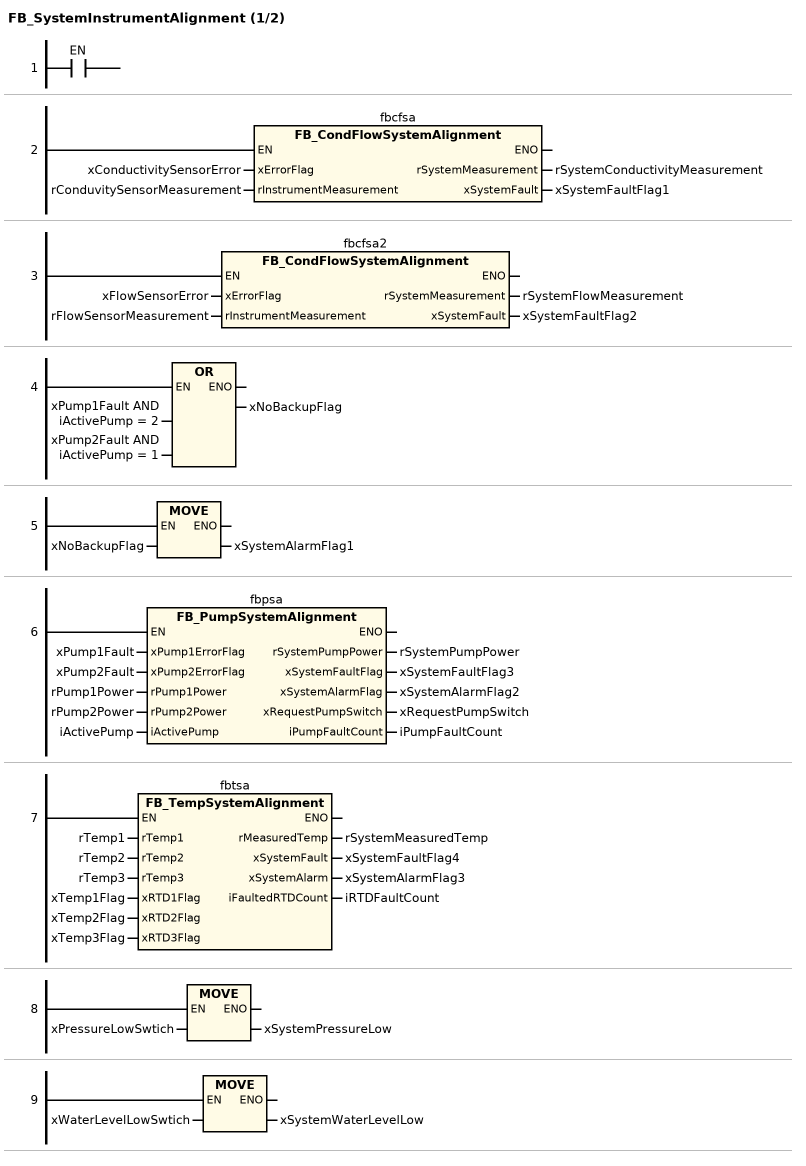
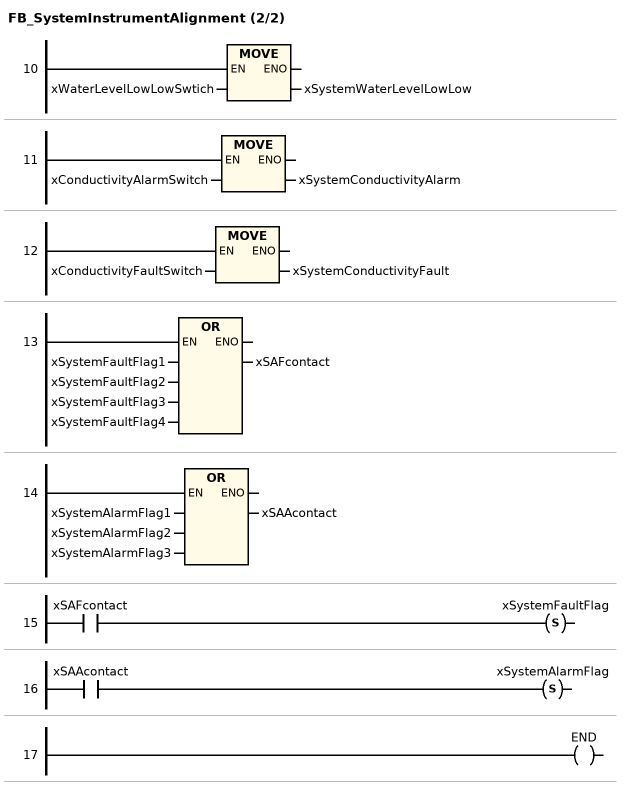
_LD_ (* Ladder Diagram *)
NETWORK 1
	[EN]
NETWORK 2
	*
		EN --- fbcfsa:FB_CondFlowSystemAlignment(xErrorFlag: xConductivitySensorError, rInstrumentMeasurement: rConduvitySensorMeasurement, xSystemFault => xSystemFaultFlag1) => rSystemConductivityMeasurement
NETWORK 3
	*
		EN --- fbcfsa2:FB_CondFlowSystemAlignment(xErrorFlag: xFlowSensorError, rInstrumentMeasurement: rFlowSensorMeasurement, xSystemFault => xSystemFaultFlag2) => rSystemFlowMeasurement
NETWORK 4
	*
		EN --- OR(xPump1Fault AND iActivePump = 2, xPump2Fault AND iActivePump = 1) => xNoBackupFlag
NETWORK 5
	*
		EN --- MOVE(xNoBackupFlag) => xSystemAlarmFlag1
NETWORK 6
	*
		EN --- fbpsa:FB_PumpSystemAlignment(xPump1ErrorFlag: xPump1Fault, xPump2ErrorFlag: xPump2Fault, rPump1Power: rPump1Power, rPump2Power: rPump2Power, iActivePump: iActivePump, xSystemFaultFlag => xSystemFaultFlag3, xSystemAlarmFlag => xSystemAlarmFlag2, xRequestPumpSwitch => xRequestPumpSwitch, iPumpFaultCount => iPumpFaultCount) => rSystemPumpPower
NETWORK 7
	*
		EN --- fbtsa:FB_TempSystemAlignment(rTemp1: rTemp1, rTemp2: rTemp2, rTemp3: rTemp3, xRTD1Flag: xTemp1Flag, xRTD2Flag: xTemp2Flag, xRTD3Flag: xTemp3Flag, xSystemFault => xSystemFaultFlag4, xSystemAlarm => xSystemAlarmFlag3, iFaultedRTDCount => iRTDFaultCount) => rSystemMeasuredTemp
NETWORK 8
	*
		EN --- MOVE(xPressureLowSwtich) => xSystemPressureLow
NETWORK 9
	*
		EN --- MOVE(xWaterLevelLowSwtich) => xSystemWaterLevelLow
NETWORK 10
	*
		EN --- MOVE(xWaterLevelLowLowSwtich) => xSystemWaterLevelLowLow
NETWORK 11
	*
		EN --- MOVE(xConductivityAlarmSwitch) => xSystemConductivityAlarm
NETWORK 12
	*
		EN --- MOVE(xConductivityFaultSwitch) => xSystemConductivityFault
NETWORK 13
	*
		EN --- OR(xSystemFaultFlag1, xSystemFaultFlag2, xSystemFaultFlag3, xSystemFaultFlag4) => xSAFcontact
NETWORK 14
	*
		EN --- OR(xSystemAlarmFlag1, xSystemAlarmFlag2, xSystemAlarmFlag3) => xSAAcontact
NETWORK 15
	[xSAFcontact] --- (S xSystemFaultFlag)
NETWORK 16
	[xSAAcontact] --- (S xSystemAlarmFlag)
NETWORK 17
	* --- (END)
_END_LD_
(* the same logic as Structured Text *)
(* Network 1 *)
(* Network 2 *)
fbcfsa(xErrorFlag := xConductivitySensorError, rInstrumentMeasurement := rConduvitySensorMeasurement);
xSystemFaultFlag1 := fbcfsa.xSystemFault;
rSystemConductivityMeasurement := fbcfsa.rSystemMeasurement;
(* Network 3 *)
fbcfsa2(xErrorFlag := xFlowSensorError, rInstrumentMeasurement := rFlowSensorMeasurement);
xSystemFaultFlag2 := fbcfsa2.xSystemFault;
rSystemFlowMeasurement := fbcfsa2.rSystemMeasurement;
(* Network 4 *)
xNoBackupFlag := (xPump1Fault AND iActivePump = 2) OR (xPump2Fault AND iActivePump = 1);
(* Network 5 *)
xSystemAlarmFlag1 := xNoBackupFlag;
(* Network 6 *)
fbpsa(xPump1ErrorFlag := xPump1Fault, xPump2ErrorFlag := xPump2Fault, rPump1Power := rPump1Power, rPump2Power := rPump2Power, iActivePump := iActivePump);
xSystemFaultFlag3 := fbpsa.xSystemFaultFlag;
xSystemAlarmFlag2 := fbpsa.xSystemAlarmFlag;
xRequestPumpSwitch := fbpsa.xRequestPumpSwitch;
iPumpFaultCount := fbpsa.iPumpFaultCount;
rSystemPumpPower := fbpsa.rSystemPumpPower;
(* Network 7 *)
fbtsa(rTemp1 := rTemp1, rTemp2 := rTemp2, rTemp3 := rTemp3, xRTD1Flag := xTemp1Flag, xRTD2Flag := xTemp2Flag, xRTD3Flag := xTemp3Flag);
xSystemFaultFlag4 := fbtsa.xSystemFault;
xSystemAlarmFlag3 := fbtsa.xSystemAlarm;
iRTDFaultCount := fbtsa.iFaultedRTDCount;
rSystemMeasuredTemp := fbtsa.rMeasuredTemp;
(* Network 8 *)
xSystemPressureLow := xPressureLowSwtich;
(* Network 9 *)
xSystemWaterLevelLow := xWaterLevelLowSwtich;
(* Network 10 *)
xSystemWaterLevelLowLow := xWaterLevelLowLowSwtich;
(* Network 11 *)
xSystemConductivityAlarm := xConductivityAlarmSwitch;
(* Network 12 *)
xSystemConductivityFault := xConductivityFaultSwitch;
(* Network 13 *)
xSAFcontact := xSystemFaultFlag1 OR xSystemFaultFlag2 OR xSystemFaultFlag3 OR xSystemFaultFlag4;
(* Network 14 *)
xSAAcontact := xSystemAlarmFlag1 OR xSystemAlarmFlag2 OR xSystemAlarmFlag3;
(* Network 15 *)
IF xSAFcontact THEN xSystemFaultFlag := TRUE; END_IF;
(* Network 16 *)
IF xSAAcontact THEN xSystemAlarmFlag := TRUE; END_IF;
(* Network 17 *)
END := TRUE;
END_FUNCTION_BLOCK

(* POU Data Conversion/Instrument->System/FB_CondFlowSystemAlignment, ST *)
FUNCTION_BLOCK FB_CondFlowSystemAlignment
VAR_INPUT
	xErrorFlag: BOOL;
	rInstrumentMeasurement: REAL;
END_VAR
VAR_OUTPUT
	rSystemMeasurement: REAL;
	xSystemFault: BOOL;
END_VAR
VAR
	rLastRead: REAL := 0;
END_VAR
IF xErrorFlag = TRUE THEN
	rSystemMeasurement := rLastRead;
	xSystemFault := TRUE;
ELSE
	rSystemMeasurement := rInstrumentMeasurement;
	rLastRead := rInstrumentMeasurement;
END_IF
END_FUNCTION_BLOCK

(* POU Data Conversion/Instrument->System/FB_PumpSystemAlignment, ST *)
FUNCTION_BLOCK FB_PumpSystemAlignment
VAR_INPUT

	xPump1ErrorFlag: BOOL;
	xPump2ErrorFlag: BOOL;
	rPump1Power: REAL;
	rPump2Power: REAL;
	iActivePump: INT;
END_VAR
VAR_OUTPUT
	rSystemPumpPower: REAL;

	xSystemFaultFlag: BOOL;
	xSystemAlarmFlag: BOOL;
	xRequestPumpSwitch: BOOL;
	iPumpFaultCount: INT;
END_VAR
VAR
	rLastPumpPowerRead: REAL;
END_VAR
VAR_IN_OUT

END_VAR
iPumpFaultCount := BOOL_TO_INT(xPump1ErrorFlag) + BOOL_TO_INT(xPump2ErrorFlag);
IF (xPump1ErrorFlag AND xPump2ErrorFlag) THEN
	xSystemFaultFlag := TRUE;
	xRequestPumpSwitch := TRUE;
ELSIF (xPump1ErrorFlag AND iActivePump = 1) OR (xPump2ErrorFlag AND iActivePump = 2) THEN
	rSystemPumpPower := rLastPumpPowerRead;
	xSystemAlarmFlag := TRUE;
	xRequestPumpSwitch := TRUE;
ELSIF iActivePump = 0 THEN
	xRequestPumpSwitch := TRUE;
	rSystemPumpPower := 0;
ELSIF iActivePump = 1 THEN
	rLastPumpPowerRead := rSystemPumpPower;
	rSystemPumpPower := rPump1Power;
ELSIF iActivePump = 2 THEN
	rLastPumpPowerRead := rSystemPumpPower;
	rSystemPumpPower := rPump2Power;
	END_IF
END_FUNCTION_BLOCK

(* POU Data Conversion/Instrument->System/FB_TempSystemAlignment, ST *)
FUNCTION_BLOCK FB_TempSystemAlignment
VAR_INPUT
	rTemp1: REAL;
	rTemp2: REAL;
	rTemp3: REAL;
	xRTD1Flag: BOOL;
	xRTD2Flag: BOOL;
	xRTD3Flag: BOOL;
END_VAR
VAR_OUTPUT
	rMeasuredTemp: REAL;
	xSystemFault: BOOL;
	xSystemAlarm: BOOL;
	iFaultedRTDCount: INT;
END_VAR
VAR
	badRTD: INT;
	rLastMeasuredValue: REAL;
END_VAR
VAR RETAIN
END_VAR
badRTD := BOOL_TO_INT(xRTD1Flag) + BOOL_TO_INT(xRTD2Flag) + BOOL_TO_INT(xRTD3Flag);
iFaultedRTDCount := badRTD;
CASE badRTD OF
	0:
		rMeasuredTemp := F_Median(rTemp1, rTemp2, rTemp3);
		rLastMeasuredValue := F_Median(rTemp1, rTemp2, rTemp3);
	1:
		rMeasuredTemp := F_AverageTemps(rTemp1, rTemp2, rTemp3, xRTD1Flag, xRTD2Flag, xRTD3Flag);
		rLastMeasuredValue := F_AverageTemps(rTemp1, rTemp2, rTemp3, xRTD1Flag, xRTD2Flag, xRTD3Flag);
		xSystemAlarm := TRUE;
	ELSE
		rMeasuredTemp := rLastMeasuredValue;
		xSystemFault := TRUE;
		xSystemAlarm := TRUE;
END_CASE
END_FUNCTION_BLOCK

(* POU Functions/F_Median, ST *)
FUNCTION F_Median : REAL
VAR_INPUT
	rValue1: REAL;
	rValue2: REAL;
	rValue3: REAL;
END_VAR
VAR
END_VAR
F_Median := MAX(MIN(rValue1, rValue2), MIN(MAX(rValue1, rValue2), rValue3));
END_FUNCTION

(* POU Functions/F_AverageTemps, ST *)
FUNCTION F_AverageTemps : REAL
VAR_INPUT
	rValue1: REAL;
	rValue2: REAL;
	rValue3: REAL;
	xTemp1Status: BOOL;
	xTemp2Status: BOOL;
	xTemp3Status: BOOL;
END_VAR
VAR
END_VAR
IF xTemp1Status = TRUE THEN
	F_AverageTemps := (rValue2 + rValue3)/2;
ELSIF xTemp2Status = TRUE THEN
	F_AverageTemps := (rValue1 + rValue3)/2;
ELSIF xTemp3Status = TRUE THEN
	F_AverageTemps := (rValue1 + rValue2)/2;
END_IF
END_FUNCTION

(* POU Instrument Control/Check Control/FB_CheckWaterLevel, ST *)
FUNCTION_BLOCK FB_CheckWaterLevel
VAR_INPUT
	EN: BOOL;
	xWaterLow: BOOL;
	xWaterVeryLow: BOOL;
END_VAR
VAR_OUTPUT
	END: BOOL;
	xSystemWaterLowFlag: BOOL;
	xSystemWaterVeryLowFlag: BOOL;
	xSystemAlarmFlag: BOOL;
	xSystemFaultFlag: BOOL;
	xWaterLevelSensorError: BOOL;

END_VAR
VAR
END_VAR
END := FALSE;
IF EN = FALSE THEN
	RETURN;
END_IF


IF xWaterLow AND xWaterVeryLow = FALSE THEN
	xSystemAlarmFlag := TRUE;
	xSystemWaterLowFlag := TRUE;
	xWaterLevelSensorError := FALSE;
ELSIF xWaterVeryLow AND xWaterLow THEN
	xSystemFaultFlag := TRUE;
	xSystemAlarmFlag := TRUE;
	xSystemWaterVeryLowFlag := TRUE;
	xWaterLevelSensorError := FALSE;
ELSIF xWaterVeryLow AND xWaterLow <> TRUE THEN
	xSystemFaultFlag := TRUE;
	xSystemAlarmFlag := TRUE;
	xWaterLevelSensorError := TRUE;
ELSE
	xSystemWaterVeryLowFlag := FALSE;
	xSystemWaterLowFlag := FALSE;
	xWaterLevelSensorError := FALSE;
END_IF

END := TRUE;
END_FUNCTION_BLOCK

(* POU Instrument Control/Check Control/FB_CheckConductivity, ST *)
FUNCTION_BLOCK FB_CheckConductivity
VAR_INPUT
	EN: BOOL;
	xConductivityBadRead: BOOL;
	xConductivityAlarmTrip: BOOL;
	xConductivityFaultTrip: BOOL;
	rConductivityMeasurement: REAL;
	rConductivityAlarmThreshold: REAL;
	rConductivityFaultThreshold: REAL;

	tHysteresisTime: TIME;
	tAlignmentTime: TIME;
END_VAR
VAR_OUTPUT
	END: BOOL;
	xConductivityMisalignmentError: BOOL;
	xConductivitySensorError: BOOL;
	xSystemAlarmFlag: BOOL;
	xSystemFaultFlag: BOOL;
	xConductivityWarning: BOOL;
	xConductivityAlert: BOOL;
END_VAR
VAR
	xConductivityAlarmBasedOnCalculations: BOOL;
	xConductivityFaultBasedOnCalculations: BOOL;
	iAlarmCount: INT;
	iFaultCount: INT;
	fbTON1: TON;
	fbTON2: TON;
	fbdebounce1: FB_DebounceSignal;
	fbdebounce2: FB_DebounceSignal;
	xConductivityMisalignmentErrorCandidate: BOOL;
END_VAR
END := FALSE;
IF EN = FALSE THEN
	RETURN;
END_IF

IF xConductivityBadRead THEN
	RETURN;
ELSE
	xConductivityAlarmBasedOnCalculations := F_BoundCheck(rInput := rConductivityMeasurement,
																	   xMaxCheck := TRUE,
																	   xMinCheck := FALSE,
																	   rMaxVariable :=  rConductivityAlarmThreshold,
																	   rMinVariable := 0,
																	   rTolerance := 0);
	fbdebounce1(EN := TRUE, xInput := xConductivityAlarmBasedOnCalculations, tDebounceTime := tHysteresisTime);

	xConductivityFaultBasedOnCalculations := F_BoundCheck(rInput := rConductivityMeasurement,
																	   xMaxCheck := TRUE,
																	   xMinCheck := FALSE,
																	   rMaxVariable :=  rConductivityFaultThreshold,
																	   rMinVariable := 0,
																	   rTolerance := 0);
	fbdebounce2(EN := TRUE, xInput := xConductivityFaultBasedOnCalculations, tDebounceTime := tHysteresisTime);

	iAlarmCount := BOOL_TO_INT(fbdebounce1.xOutput) + BOOL_TO_INT(xConductivityAlarmTrip);
	iFaultCount := BOOL_TO_INT(fbdebounce2.xOutput) + BOOL_TO_INT(xConductivityFaultTrip);

	IF iAlarmCount = 1 OR iFaultCount = 1 THEN
		xConductivityMisalignmentErrorCandidate := TRUE;
	END_IF
	IF (iFaultCount = 2 AND iAlarmCount = 1) THEN (*This guarantees that the sensor is not working*)
		xConductivitySensorError := TRUE;
		xSystemFaultFlag := TRUE;
	END_IF
	IF (iFaultCount = 2 AND iAlarmCount = 2) OR (iAlarmCount = 2) OR (iFaultCount = 0 AND iAlarmCount = 0) THEN
		xConductivityMisalignmentErrorCandidate := FALSE;
		xConductivitySensorError := FALSE;
	END_IF
	IF iAlarmCount = 2 THEN
		xSystemAlarmFlag := TRUE;
		xConductivityWarning := TRUE;
	ELSIF iAlarmCount= 0 THEN
		xConductivityWarning := FALSE;
	END_IF
	IF iFaultCount = 2 THEN
		xSystemFaultFlag := TRUE;
		xConductivityAlert := TRUE;
	ELSIF iFaultCount = 0 THEN
		xConductivityAlert := FALSE;
	END_IF
END_IF
fbTON1(IN := xConductivityMisalignmentErrorCandidate, PT := tAlignmentTime);

IF fbTON1.Q THEN
	xConductivityMisalignmentError := TRUE;
	xSystemFaultFlag := TRUE;
ELSE
	xConductivityMisalignmentError := FALSE;
END_IF
END := TRUE;
END_FUNCTION_BLOCK

(* POU Instrument Control/Check Control/FB_PowerPressureFlowThreshold, ST *)
FUNCTION_BLOCK FB_PowerPressureFlowThreshold
VAR_INPUT
	EN: BOOL;
	rPumpPowerLowThreshold: REAL;
	rPumpPower: REAL;
	rFlow: REAL;
	rFlowLowThreshold: REAL;
	xPressureLowInput: BOOL;
	tHysteresisTime: TIME;
END_VAR
VAR_OUTPUT
	END: BOOL;
	xPumpPowerLow: BOOL;
	xFlowLow: BOOL;
	xPressureLowFlag: BOOL;
END_VAR
VAR
	fbInitializeTimer: TON;
	xPumpPowerLowUF: BOOL;
	fbTON1: TON;
	xFlowLowUF: BOOL;
	fbTON2: TON;
	fbdebounce1: FB_DebounceSignal;
	fbdebounce2: FB_DebounceSignal;
END_VAR
IF EN = FALSE THEN
	RETURN;
END_IF
END := FALSE;
xPumpPowerLowUF := F_BoundCheck(rInput := rPumpPower,
										 xMaxCheck := FALSE,
										 xMinCheck := TRUE,
										 rMaxVariable :=  0,
										 rMinVariable := rPumpPowerLowThreshold,
										 rTolerance := 0);
fbdebounce1(EN := TRUE, xInput := xPumpPowerLowUF, tDebounceTime := tHysteresisTime);
xPumpPowerLow := fbdebounce1.xOutput;

xFlowLowUF := F_BoundCheck(rInput := rFlow,
										 xMaxCheck := FALSE,
										 xMinCheck := TRUE,
										 rMaxVariable :=  0,
										 rMinVariable := rFlowLowThreshold,
										 rTolerance := 0);
fbdebounce2(EN := TRUE, xInput := xFlowLowUF, tDebounceTime := tHysteresisTime);
xFlowLow := fbdebounce2.xOutput;


xPressureLowFlag := xPressureLowInput;

END := TRUE;
END_FUNCTION_BLOCK

(* POU Instrument Control/Check Control/FB_PowerPressureFlowVote, ST *)
FUNCTION_BLOCK FB_PowerPressureFlowVote
VAR_INPUT
	EN: BOOL;
	xLowPressure: BOOL;
	xLowFlow: BOOL;
	xLowPower: BOOL;
	xNoBackupFlag: BOOL;
	iActivePump: INT;
	xAwaitSystemInit: BOOL;
END_VAR
VAR_OUTPUT
	END: BOOL;
	xSystemFaultFlag: BOOL;
	xSystemAlarmFlag: BOOL;
	xRequestPumpSwitch: BOOL;
	xPPFError: BOOL;
	xPump1LPError: BOOL;
	xPump2LPError: BOOL;
END_VAR
VAR
	iBadCount: INT;
END_VAR
IF EN = FALSE THEN
	RETURN;
END_IF
END := FALSE;
iBadCount := BOOL_TO_INT(xLowPressure) + BOOL_TO_INT(xLowFlow) + BOOL_TO_INT(xLowPower);

IF xAwaitSystemInit OR iActivePump = 0 THEN
	RETURN;
ELSE
	IF iBadCount = 1 THEN
		xSystemAlarmFlag := TRUE;
	ELSIF  (iBadCount > 1) THEN
		xRequestPumpSwitch := TRUE;
		xPPFError := TRUE;
		IF xNoBackupFlag = TRUE THEN
			xSystemFaultFlag := TRUE;
		END_IF
	END_IF
	IF iActivePump = 1 THEN
		xPump1LPError := xLowPower;
	ELSIF iActivePump = 2 THEN
		xPump2LPError := xLowPower;
	END_IF
END_IF
END := TRUE;
END_FUNCTION_BLOCK

(* POU Instrument Control/FB_PumpStartSwitchRoutine, ST *)
FUNCTION_BLOCK FB_PumpStartSwitchRoutine
VAR_INPUT
	EN: BOOL;
	iActiveNumberOfPumps: INT;
	xPump1FailFlag: BOOL;
	xPump2FailFlag: BOOL;
	xPump1LPFlag: BOOL;
	xPump2LPFlag: BOOL;
	xPPFError: BOOL;
	tDebouceTimeDoubled: TIME;
END_VAR
VAR_OUTPUT
	END: BOOL;
	xPump1ActuationVariable: BOOL;
	xPump2ActuationVariable: BOOL;
	xSystemAlarm: BOOL;
	xSystemFault: BOOL;
END_VAR
VAR
	fbbypass: TON;
END_VAR
VAR_IN_OUT
	xNoBackupFlag: BOOL;
	xRequestPumpSwitch: BOOL;
	xAwaitSystemInit: BOOL;
END_VAR
fbbypass(IN := TRUE,  PT := tDebouceTimeDoubled);
IF EN = FALSE OR fbbypass.Q = FALSE  THEN
	RETURN;
END_IF
END := FALSE;
IF xRequestPumpSwitch AND xNoBackupFlag THEN
	xSystemFault := TRUE;
	xPump1ActuationVariable := FALSE;
	xPump2ActuationVariable := FALSE;
ELSIF xRequestPumpSwitch AND xNoBackupFlag = FALSE AND xAwaitSystemInit = FALSE THEN
	xAwaitSystemInit := TRUE;
	CASE  iActiveNumberOfPumps OF
		0:
			IF (xPump1FailFlag OR xPump1LPFlag) THEN
				xPump1ActuationVariable := FALSE;
				xPump2ActuationVariable := TRUE;
			ELSIF (xPump1FailFlag = FALSE OR xPump1LPFlag = FALSE) THEN
				xPump1ActuationVariable := TRUE;
				xPump2ActuationVariable := FALSE;
			END_IF
		1:
			xPump1ActuationVariable := FALSE;
			xPump2ActuationVariable := TRUE;
			IF (xPump1FailFlag OR (xPump1LPFlag AND xPPFError)) THEN
				xNoBackupFlag := TRUE;
				xSystemAlarm := TRUE;
			END_IF
		2:
			xPump1ActuationVariable := TRUE;
			xPump2ActuationVariable := FALSE;
			IF (xPump2FailFlag OR (xPump2LPFlag AND xPPFError)) THEN
				xNoBackupFlag := TRUE;
				xSystemAlarm := TRUE;
			END_IF
		ELSE
			xSystemFault := TRUE;
			xPump1ActuationVariable := FALSE;
			xPump2ActuationVariable := FALSE;
			xNoBackupFlag := TRUE;
	END_CASE
END_IF
xRequestPumpSwitch := FALSE;
END := TRUE;
END_FUNCTION_BLOCK

(* POU Instrument Control/Check Control/FB_TemperatureBoundCheck, ST *)
FUNCTION_BLOCK FB_TemperatureBoundCheck
VAR_INPUT
	EN: BOOL;
	rSystemTemperature: REAL;
	rTempFaultMin: REAL;
	rTempFaultMax: REAL;
	rTempAlarmMin: REAL;
	rTempAlarmMax: REAL;
	tWarningTime: TIME;
	tFailureTime: TIME;
	xAwaitInit: BOOL;
	xAwaitCalibration: BOOL;
	xStartDelay: BOOL;
END_VAR
VAR_OUTPUT
	END: BOOL;
	xTemperatureWarning: BOOL;
	xTemperatureFailure: BOOL;
END_VAR
VAR
	xTempAlarm: BOOL;
	xTempFault: BOOL;
	fbTON1: TON;
	fbTON2: TON;
END_VAR
END := FALSE;
IF xAwaitInit OR xAwaitCalibration OR xStartDelay OR EN = FALSE THEN
	RETURN;
ELSE
	xTempAlarm := F_BoundCheck(rInput := rSystemTemperature,
										 	xMaxCheck := TRUE,
										 	xMinCheck := TRUE,
										 	rMaxVariable :=  rTempAlarmMin,
										 	rMinVariable := rTempAlarmMax,
										 	rTolerance := 0);
	xTempFault := F_BoundCheck(rInput := rSystemTemperature,
										 	xMaxCheck := TRUE,
										 	xMinCheck := TRUE,
										 	rMaxVariable :=  rTempFaultMin,
										 	rMinVariable := rTempFaultMax,
										 	rTolerance := 0);

END_IF
fbTON1(IN := xTempAlarm, PT := tWarningTime);
fbTON2(IN := xTempFault, PT := tFailureTime);
xTemperatureWarning := fbTON1.Q;
xTemperatureFailure := fbTON2.Q;
END_FUNCTION_BLOCK

(* POU System Startup/FB_SystemStart, ST *)
FUNCTION_BLOCK FB_SystemStart
VAR_INPUT
	xEnable: BOOL;

	tInitilizationTime: TIME;
	tCalibrationTime: TIME;
	xSystemShutdownInProgress: BOOL;
END_VAR
VAR_OUTPUT
	xDone: BOOL;

END_VAR
VAR
	i: INT;

	fbInit: TON;
	fbCali: TON;
END_VAR
VAR_IN_OUT
	xBeginSystemInitialization: BOOL;
	axInstrumentFlags: ARRAY [1..25] OF BOOL;
	xSystemOn: BOOL;
	xFaultACK: BOOL;
	xFaultExists: BOOL;
	xSystemInitializing: BOOL;
	xSystemCalibrating: BOOL;
END_VAR
xDone := FALSE;
IF xEnable = FALSE THEN
	RETURN;
END_IF;

fbInit(IN := xSystemOn, PT := tInitilizationTime);
fbCali(IN:= fbInit.Q, PT := tCalibrationTime);

IF (xSystemShutdownInProgress = TRUE) OR (xBeginSystemInitialization = TRUE AND xFaultExists = TRUE AND xFaultAck = FALSE) OR (xBeginSystemInitialization = TRUE AND xFaultExists = FALSE AND xFaultAck = TRUE)  THEN
	xBeginSystemInitialization := FALSE;
	RETURN;
ELSIF (xBeginSystemInitialization = TRUE AND xFaultExists = TRUE AND xFaultACK = TRUE) THEN
	FOR i := 1 TO 25 DO
		axInstrumentFlags[i] := FALSE;
	END_FOR;
	xSystemOn := TRUE;
	xSystemInitializing := TRUE;
	xSystemCalibrating := TRUE;
	xBeginSystemInitialization := FALSE;
	xFaultExists := FALSE;
	xFaultACK := FALSE;
ELSIF xBeginSystemInitialization = TRUE AND xFaultExists = FALSE AND xFaultACK = FALSE THEN
	xSystemOn := TRUE;
	xSystemInitializing := TRUE;
	xSystemCalibrating := TRUE;
	xBeginSystemInitialization := FALSE;
END_IF

IF fbInit.Q = TRUE THEN
	xSystemInitializing := FALSE;
END_IF
IF fbCali.Q = TRUE THEN
	xSystemCalibrating := FALSE;
END_IF

xDone := TRUE;
END_FUNCTION_BLOCK

(* POU System Startup/FB_FaultCheck, ST *)
FUNCTION_BLOCK FB_FaultCheck
VAR_INPUT
	xEnable: BOOL;
	axInstrumentFlags: ARRAY [1..25] OF BOOL;
END_VAR
VAR_OUTPUT
	xDone: BOOL;

END_VAR
VAR
	i: INT;
END_VAR
VAR_IN_OUT
	xFaultExists: BOOL;
END_VAR
xDone := FALSE;
IF xEnable = FALSE THEN
	RETURN;
END_IF;
FOR i := 1 TO 15 DO
		IF axInstrumentFlags[i] = TRUE THEN
			xFaultExists := TRUE;
		END_IF;
END_FOR;
xDone := TRUE;
END_FUNCTION_BLOCK

(* POU System Startup/FB_SystemStop, ST *)
FUNCTION_BLOCK FB_SystemStop
VAR_INPUT
	xEnable: BOOL;

	xFaultExists: BOOL;
	tSDTime: TIME;
END_VAR
VAR_OUTPUT
	xDone: BOOL;

END_VAR
VAR
	xOFF: BOOL;
	fbSD: TON;

END_VAR

VAR_IN_OUT
	xSystemShutdownInProgress: BOOL;
	xSystemOn: BOOL;
	xSystemInitializing: BOOL;
	xSystemCalibrating: BOOL;
	xForceShutdown: BOOL;
END_VAR
xDone := FALSE;
IF xEnable = FALSE THEN
	RETURN;
END_IF
fbSD(IN := 	xSystemShutdownInProgress, PT := tSDTime);
IF (xForceShutdown = FALSE AND xFaultExists = FALSE AND xSystemShutdownInProgress = FALSE AND xSystemOn = TRUE) OR xSystemOn = FALSE THEN
	RETURN;
ELSIF (xForceShutdown = TRUE OR xFaultExists = TRUE) AND (xSystemShutdownInProgress = FALSE) THEN
	xForceShutdown := FALSE;
	xSystemShutdownInProgress := TRUE;
	xSystemInitializing := FALSE;
	xSystemCalibrating := FALSE;
END_IF



IF fbSD.Q THEN
	xSystemShutdownInProgress := FALSE;
	xSystemOn := FALSE;
END_IF
xDone := TRUE;
END_FUNCTION_BLOCK

(* POU Instrument Control/FB_PumpControl, ST *)
FUNCTION_BLOCK FB_PumpControl
VAR_INPUT
	EN: BOOL;
	xSystemShutdownInProgress: BOOL;
	xSystemON: BOOL;
	xSimplex: BOOL;
END_VAR
VAR_OUTPUT
	END: BOOL;

END_VAR
VAR
END_VAR
VAR_IN_OUT
	xPrimaryPumpActive: BOOL;
	xSecondaryPumpActive: BOOL;
	xAutohandover: BOOL;
	xManualhandover: BOOL;
END_VAR
END := FALSE;
IF EN = FALSE THEN
	RETURN;
END_IF
IF (xSystemShutdownInProgress = TRUE OR xSystemON = FALSE) THEN
	xPrimaryPumpActive := FALSE;
	xSecondaryPumpActive := FALSE;
ELSIF xSystemON = TRUE AND xSystemShutdownInProgress = FALSE AND xPrimaryPumpActive = FALSE AND xSecondaryPumpActive = FALSE AND (xAutohandover OR (xManualhandover AND xSimplex = FALSE)) THEN
	xPrimaryPumpActive := TRUE;
	xSecondaryPumpActive := FALSE;
ELSIF xSystemON = TRUE AND xSystemShutdownInProgress = FALSE AND xPrimaryPumpActive = FALSE AND xSecondaryPumpActive = TRUE AND (xAutohandover OR (xManualhandover AND xSimplex = FALSE))  THEN
	xPrimaryPumpActive := TRUE;
	xSecondaryPumpActive := FALSE;
ELSIF xSystemON = TRUE AND xSystemShutdownInProgress = FALSE AND xPrimaryPumpActive = FALSE AND xSecondaryPumpActive = TRUE AND (xAutohandover OR (xManualhandover AND xSimplex = FALSE))  THEN
	xPrimaryPumpActive := FALSE;
	xSecondaryPumpActive := TRUE;
END_IF
xAutohandover = FALSE;
xManualhandover = FALSE;
END := TRUE;
END_FUNCTION_BLOCK

(* POU Legacy/FB_DigitalCapture, ST *)
FUNCTION_BLOCK FB_DigitalCapture
VAR_INPUT

	xEnable: BOOL;		(*Activates Function Block*)
	xRawInput: BOOL;
	tDebounceTime: TIME := T#50MS;		(*How long do you want to wait until it reaches a stable state*)
	xRisingEdgeDetection: BOOL; (*Is this something where we just want to measure the instance it turns on? Like user input*)
	xFallingEdgeDetection: BOOL; (*|| but off*)

END_VAR
VAR_OUTPUT
	xContinue: BOOL := TRUE;
	xRisingEdgeDetected: BOOL;
	xFallingEdgeDetected: BOOL;
END_VAR
VAR
	xRawDigitalInput: BOOL;		(*Raw Input Value from Instrument*)
	fbDebounceTimerON:TON;
	fbDebounceTimerOFF: TOF;
	fbRisingEdge: R_TRIG;
	fbFallingEdge: F_TRIG;
	iCheck: INT;
END_VAR
VAR_IN_OUT
	stInstrument: ST_INSTRUMENT;		(*User Defined Instrument*)
END_VAR
(*This takes raw digital input and stores it in instrumentation data*)
(*We need to check if 	), b) ensure hystersis does not occur (like analog), c) check if this is a user input (edge detection, versus just on/off*)

IF xEnable = FALSE THEN (*Check if we're enabled*)
	RETURN;
END_IF

(*
fbDebounceTimerON(IN := xRawInput, PT := tDebounceTime); (*Won't go to true until 50 ms of stability. Every false resets this timer*)
fbDebounceTimerOFF(IN := fbDebounceTimerON.Q, PT := tDebounceTime); (*Won't go to false until 50ms of stability. Every true resets this timer*)

xRawDigitalInput := fbDebounceTimerOFF.Q;
stInstrument.xCapturedBoolSignal := xRawDigitalInput;
fbRisingEdge(CLK := xRawDigitalInput);
fbFallingEdge(CLK := xRawDigitalInput);
IF xRisingEdgeDetection = TRUE AND xFallingEdgeDetection = TRUE THEN
	stInstrument.xCapturedBoolValue := fbRisingEdge.Q OR fbFallingEdge.Q; (*Are we detecing if this goes from False to True. When we detect this, caputre it*)
	IF (stInstrument.xCapturedBoolValue = TRUE) THEN
		iCheck := iCheck + 1;
	END_IF
ELSIF xFallingEdgeDetection = TRUE THEN
	stInstrument.xCapturedBoolValue := fbFallingEdge.Q; (*Same as above but Vice Versa. Note that you can have both!*)
	IF (stInstrument.xCapturedBoolValue = TRUE) THEN
		iCheck := iCheck + 1;
		xFallingEdgeDetected := TRUE;
	END_IF
ELSIF xRisingEdgeDetection = TRUE THEN
	stInstrument.xCapturedBoolValue := fbRisingEdge.Q;
	IF (stInstrument.xCapturedBoolValue = TRUE) THEN
		iCheck := iCheck + 1;
		xRisingEdgeDetected := TRUE;
	END_IF
ELSE
	stInstrument.xCapturedBoolValue := stInstrument.xCapturedBoolSignal;
END_IF


*)
END_FUNCTION_BLOCK

(* POU Test Bench Folder/TB_CalibrationClock, LD *)
PROGRAM TB_CalibrationClock
VAR
	a: BOOL;
	b: BOOL;
	fbct: FB_CalibrationTimer;
END_VAR
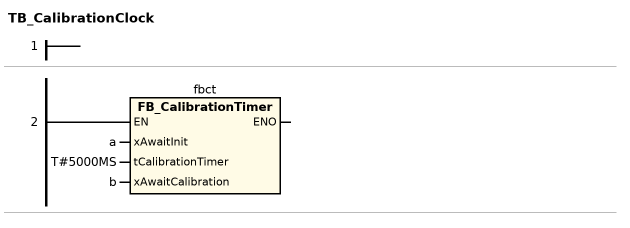
_LD_ (* Ladder Diagram *)
NETWORK 1
	*
NETWORK 2
	*
		EN --- fbct:FB_CalibrationTimer(xAwaitInit: a, tCalibrationTimer: T#5000MS, xAwaitCalibration: b)
_END_LD_
(* the same logic as Structured Text *)
(* Network 1 *)
(* Network 2 *)
fbct(xAwaitInit := a, tCalibrationTimer := T#5000MS, xAwaitCalibration := b);
END_PROGRAM

(* POU Instrument Control/Check Control/FB_CalibrationTimer, ST *)
FUNCTION_BLOCK FB_CalibrationTimer
VAR_INPUT
	xAwaitInit: BOOL;
	tCalibrationTimer: TIME;
END_VAR
VAR_OUTPUT
END_VAR
VAR
	xBeginClock: BOOL;
	fbTimerON: TON;
END_VAR
VAR_IN_OUT
	xAwaitCalibration: BOOL;
END_VAR
fbTimerON(IN := xBeginClock, PT := tCalibrationTimer);
IF xAwaitInit AND xAwaitCalibration = FALSE THEN
	xAwaitCalibration := TRUE;
ELSIF xAwaitInit = FALSE AND (xAwaitCalibration OR xBeginClock) THEN
	xBeginClock := TRUE;
ELSIF xAwaitInit AND xBeginClock THEN
	xBeginClock := FALSE;
	xAwaitCalibration := TRUE;
ELSIF xAwaitInit AND xAwaitCalibration THEN
	RETURN;
END_IF

IF xBeginClock = TRUE AND fbTimerON.Q = TRUE THEN
	xAwaitCalibration := FALSE;
	xBeginClock := FALSE;
END_IF
END_FUNCTION_BLOCK

(* POU Test Bench Folder/TB_CheckConductivity, LD *)
PROGRAM TB_CheckConductivity
VAR
	a: BOOL := FALSE;
	b: BOOL := FALSE;
	c: BOOL := FALSE;
	d: REAL := 4;
	e: REAL := 10;
	f: REAL := 15;
	z: BOOL;
	y: BOOL;
	x: BOOL;
	w: BOOL;
	v: BOOL;
	u: BOOL;
	fbcc: FB_CheckConductivity;
END_VAR
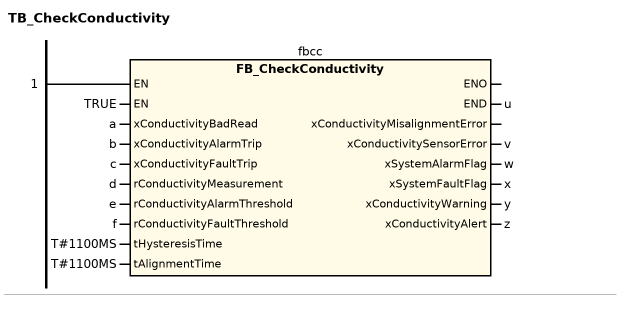
_LD_ (* Ladder Diagram *)
NETWORK 1
	*
		EN --- fbcc:FB_CheckConductivity(EN: TRUE, xConductivityBadRead: a, xConductivityAlarmTrip: b, xConductivityFaultTrip: c, rConductivityMeasurement: d, rConductivityAlarmThreshold: e, rConductivityFaultThreshold: f, tHysteresisTime: T#1100MS, tAlignmentTime: T#1100MS, xConductivitySensorError => v, xSystemAlarmFlag => w, xSystemFaultFlag => x, xConductivityWarning => y, xConductivityAlert => z) => u
_END_LD_
(* the same logic as Structured Text *)
(* Network 1 *)
fbcc(EN := TRUE, xConductivityBadRead := a, xConductivityAlarmTrip := b, xConductivityFaultTrip := c, rConductivityMeasurement := d, rConductivityAlarmThreshold := e, rConductivityFaultThreshold := f, tHysteresisTime := T#1100MS, tAlignmentTime := T#1100MS);
v := fbcc.xConductivitySensorError;
w := fbcc.xSystemAlarmFlag;
x := fbcc.xSystemFaultFlag;
y := fbcc.xConductivityWarning;
z := fbcc.xConductivityAlert;
u := fbcc.END;
END_PROGRAM

(* POU Test Bench Folder/TB_InputTest, LD *)
PROGRAM TB_InputTest
VAR
	xOnOff: BOOL;
END_VAR
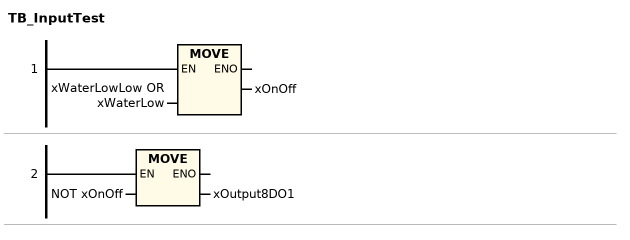
_LD_ (* Ladder Diagram *)
NETWORK 1
	*
		EN --- MOVE( xWaterLowLow OR xWaterLow) => xOnOff
NETWORK 2
	*
		EN --- MOVE(NOT xOnOff) => xOutput8DO1
_END_LD_
(* the same logic as Structured Text *)
(* Network 1 *)
xOnOff :=  xWaterLowLow OR xWaterLow;
(* Network 2 *)
xOutput8DO1 := NOT xOnOff;
END_PROGRAM

(* POU Test Bench Folder/TB_InstrumentReadErrorFaultAlignment, LD *)
PROGRAM TB_InstrumentReadErrorFaultAlignment
VAR
	pbr1: BOOL := FALSE;
	pbr2: BOOL := FALSE;
	tbr1: BOOL := FALSE;
	tbr2: BOOL := FALSE;
	tbr3: BOOL := FALSE;
	cbr: BOOL := FALSE;
	fbr: BOOL := FALSE;
	pef1: BOOL;
	pef2: BOOL;
	pef3: BOOL;
	tef1: BOOL;
	tef2: BOOL;
	tef3: BOOL;
	cef: BOOL;
	fef: BOOL;
	fbirr: FB_InstrumentReadRecon;
END_VAR
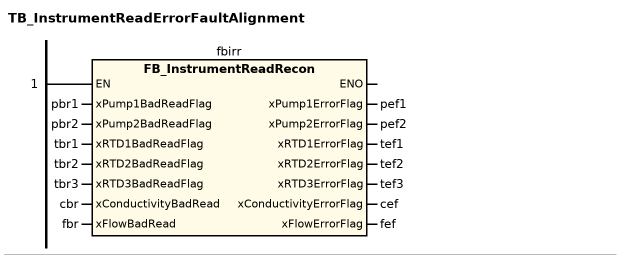
_LD_ (* Ladder Diagram *)
NETWORK 1
	*
		EN --- fbirr:FB_InstrumentReadRecon(xPump1BadReadFlag: pbr1, xPump2BadReadFlag: pbr2, xRTD1BadReadFlag: tbr1, xRTD2BadReadFlag: tbr2, xRTD3BadReadFlag: tbr3, xConductivityBadRead: cbr, xFlowBadRead: fbr, xPump2ErrorFlag => pef2, xRTD1ErrorFlag => tef1, xRTD2ErrorFlag => tef2, xRTD3ErrorFlag => tef3, xConductivityErrorFlag => cef, xFlowErrorFlag => fef) => pef1
_END_LD_
(* the same logic as Structured Text *)
(* Network 1 *)
fbirr(xPump1BadReadFlag := pbr1, xPump2BadReadFlag := pbr2, xRTD1BadReadFlag := tbr1, xRTD2BadReadFlag := tbr2, xRTD3BadReadFlag := tbr3, xConductivityBadRead := cbr, xFlowBadRead := fbr);
pef2 := fbirr.xPump2ErrorFlag;
tef1 := fbirr.xRTD1ErrorFlag;
tef2 := fbirr.xRTD2ErrorFlag;
tef3 := fbirr.xRTD3ErrorFlag;
cef := fbirr.xConductivityErrorFlag;
fef := fbirr.xFlowErrorFlag;
pef1 := fbirr.xPump1ErrorFlag;
END_PROGRAM

(* POU Data Conversion/Instrument->System/FB_InstrumentReadRecon, ST *)
FUNCTION_BLOCK FB_InstrumentReadRecon
VAR_INPUT
	xPump1BadReadFlag: BOOL;
	xPump2BadReadFlag: BOOL;
	xRTD1BadReadFlag: BOOL;
	xRTD2BadReadFlag: BOOL;
	xRTD3BadReadFlag: BOOL;
	xConductivityBadRead: BOOL;
	xFlowBadRead: BOOL;
END_VAR
VAR_OUTPUT
	xPump1ErrorFlag: BOOL;
	xPump2ErrorFlag: BOOL;
	xRTD1ErrorFlag: BOOL;
	xRTD2ErrorFlag: BOOL;
	xRTD3ErrorFlag: BOOL;
	xConductivityErrorFlag: BOOL;
	xFlowErrorFlag: BOOL;
END_VAR
VAR
END_VAR
 xPump1ErrorFlag :=  xPump1BadReadFlag;
xPump2ErrorFlag := xPump2BadReadFlag;
xRTD1ErrorFlag := xRTD1BadReadFlag;
xRTD2ErrorFlag :=  xRTD2BadReadFlag;
xRTD3ErrorFlag := xRTD3BadReadFlag;
 xConductivityErrorFlag := xConductivityBadRead;
xFlowErrorFlag := xFlowBadRead;
END_FUNCTION_BLOCK

(* POU Test Bench Folder/TB_PowerPressureFlowVote, LD *)
PROGRAM TB_PowerPressureFlowVote
VAR

